// TwinCAT 3 PLC project PLC1
// ProgramVersion: 3.1.4024.12
// libraries:
//   Tc2_EtherCAT, * (Beckhoff Automation GmbH)
//   Tc2_Standard, * (Beckhoff Automation GmbH)
//   Tc2_System, * (Beckhoff Automation GmbH)
//   Tc2_Utilities, * (Beckhoff Automation GmbH)
//   Tc3_Module, * (Beckhoff Automation GmbH)
//   VisuSymbols,3.5.10.0,System
// project tree:
//   / Class Diagram.TcCD (not stored), GlobalTextList.TcGTLO, PlcTask.TcTTO, Visualization Manager.TcVMO (not stored)
//   DUTs/ ST_1In.TcDUT, ST_1In1Out.TcDUT, ST_2In.TcDUT, ST_2Out.TcDUT, ST_EL1004.TcDUT, ST_EL1008.TcDUT, ST_EL2004.TcDUT, ST_EL2008.TcDUT
//   GVLs/ GVL_Constants.TcGVL, GVL_HMI.TcGVL, GVL_IO.TcGVL
//   POUs/FunctionBlocks/ FB_1In.TcPOU, FB_1In_1Out.TcPOU, FB_2In.TcPOU, FB_2Out.TcPOU
//   POUs/FunctionBlocks/Flow FBs/ FB_HandshakeControl.TcPOU
//   POUs/Interfaces/ I_ConveyerSection.TcIO
//   POUs/ MAIN.TcPOU
//   VISUs/ Physical.TcVIS, Configured.TcVIS, RackText.TcTLO
// real-time tasks:
//   TASK PlcTask: cycle T#10ms, priority 20, ADS port 350
//   TASK VISU_TASK: cycle T#200000us, priority 30, ADS port 351
// I/O:
//   DEVICE HotConnect Demo(EtherCAT), AmsNetId 5.29.120.74.5.1
//     2 In_1 [EK1101 EtherCAT Coupler (2A E-Bus, ID switch)]
//       Term 11 (EL1008) [EL1008 8Ch. Dig. Input 24V, 3ms]
//       Term 12 (EL1008) [EL1008 8Ch. Dig. Input 24V, 3ms]
//       Term 1 (EL7031) [EL7031 1Ch. Stepper motor output stage (24V, 1.5A)]
//     2 In_2 [EK1101 EtherCAT Coupler (2A E-Bus, ID switch)]
//       Term 14 (EL1008) [EL1008 8Ch. Dig. Input 24V, 3ms]
//       Term 15 (EL1008) [EL1008 8Ch. Dig. Input 24V, 3ms]
//     1 In 1 out_1 [EK1101 EtherCAT Coupler (2A E-Bus, ID switch)]
//       Term 18 (EL1008) [EL1008 8Ch. Dig. Input 24V, 3ms]
//       Term 19 (EL2008) [EL2008 8Ch. Dig. Output 24V, 0.5A]
//     1 in 1 out_2 [EK1101 EtherCAT Coupler (2A E-Bus, ID switch)]
//       Term 20 (EL1008) [EL1008 8Ch. Dig. Input 24V, 3ms]
//       Term 21 (EL2008) [EL2008 8Ch. Dig. Output 24V, 0.5A]
//     2 Out_1 [EK1101 EtherCAT Coupler (2A E-Bus, ID switch)]
//       Term 24 (EL2008) [EL2008 8Ch. Dig. Output 24V, 0.5A]
//       Term 25 (EL2008) [EL2008 8Ch. Dig. Output 24V, 0.5A]
//     2 Out_2 [EK1101 EtherCAT Coupler (2A E-Bus, ID switch)]
//       Term 26 (EL2008) [EL2008 8Ch. Dig. Output 24V, 0.5A]
//       Term 27 (EL2008) [EL2008 8Ch. Dig. Output 24V, 0.5A]
//     1 In_1 [EK1101 EtherCAT Coupler (2A E-Bus, ID switch)]
//       Term 30 (EL1008) [EL1008 8Ch. Dig. Input 24V, 3ms]
//     1 In_2 [EK1101 EtherCAT Coupler (2A E-Bus, ID switch)]
//       Term 31 (EL1008) [EL1008 8Ch. Dig. Input 24V, 3ms]
// variable links:
//   PLC1/PLC1 Instance <-> HotConnect Demo(EtherCAT)/1 In 1 out_1
//     PlcTask Inputs/GVL_IO.arrIds[2] <-> ID/ID
//     PlcTask Inputs/GVL_IO.arrState[2] <-> InfoData/State
//   PLC1/PLC1 Instance <-> HotConnect Demo(EtherCAT)/1 In 1 out_1/Term 18 (EL1008)
//     PlcTask Inputs/MAIN.arrFb1In1Out[0].stRack.ST_In/Input{1..8} <-> Channel {1..8}/Input  (8 links)
//   PLC1/PLC1 Instance <-> HotConnect Demo(EtherCAT)/1 In 1 out_1/Term 19 (EL2008)
//     PlcTask Outputs/MAIN.arrFb1In1Out[0].stRack.ST_Out/Output{1..8} <-> Channel {1..8}/Output  (8 links)
//   PLC1/PLC1 Instance <-> HotConnect Demo(EtherCAT)/1 In_1
//     PlcTask Inputs/GVL_IO.arrIds[6] <-> ID/ID
//     PlcTask Inputs/GVL_IO.arrState[6] <-> InfoData/State
//   PLC1/PLC1 Instance <-> HotConnect Demo(EtherCAT)/1 In_1/Term 30 (EL1008)
//     PlcTask Inputs/MAIN.arrFb1In[0].stRack.ST_In/Input{1..8} <-> Channel {1..8}/Input  (8 links)
//   PLC1/PLC1 Instance <-> HotConnect Demo(EtherCAT)/1 In_2
//     PlcTask Inputs/GVL_IO.arrIds[7] <-> ID/ID
//     PlcTask Inputs/GVL_IO.arrState[7] <-> InfoData/State
//   PLC1/PLC1 Instance <-> HotConnect Demo(EtherCAT)/1 In_2/Term 31 (EL1008)
//     PlcTask Inputs/MAIN.arrFb1In[1].stRack.ST_In/Input{1..8} <-> Channel {1..8}/Input  (8 links)
//   PLC1/PLC1 Instance <-> HotConnect Demo(EtherCAT)/1 in 1 out_2
//     PlcTask Inputs/GVL_IO.arrIds[3] <-> ID/ID
//     PlcTask Inputs/GVL_IO.arrState[3] <-> InfoData/State
//   PLC1/PLC1 Instance <-> HotConnect Demo(EtherCAT)/1 in 1 out_2/Term 20 (EL1008)
//     PlcTask Inputs/MAIN.arrFb1In1Out[1].stRack.ST_In/Input{1..8} <-> Channel {1..8}/Input  (8 links)
//   PLC1/PLC1 Instance <-> HotConnect Demo(EtherCAT)/1 in 1 out_2/Term 21 (EL2008)
//     PlcTask Outputs/MAIN.arrFb1In1Out[1].stRack.ST_Out/Output{1..8} <-> Channel {1..8}/Output  (8 links)
//   PLC1/PLC1 Instance <-> HotConnect Demo(EtherCAT)/2 In_1
//     PlcTask Inputs/GVL_IO.arrIds[0] <-> ID/ID
//     PlcTask Inputs/GVL_IO.arrState[0] <-> InfoData/State
//   PLC1/PLC1 Instance <-> HotConnect Demo(EtherCAT)/2 In_1/Term 11 (EL1008)
//     PlcTask Inputs/MAIN.arrFb2In[0].stRack.ST_in1/Input{1..8} <-> Channel {1..8}/Input  (8 links)
//   PLC1/PLC1 Instance <-> HotConnect Demo(EtherCAT)/2 In_1/Term 12 (EL1008)
//     PlcTask Inputs/MAIN.arrFb2In[0].stRack.ST_in2/Input{1..8} <-> Channel {1..8}/Input  (8 links)
//   PLC1/PLC1 Instance <-> HotConnect Demo(EtherCAT)/2 In_2
//     PlcTask Inputs/GVL_IO.arrIds[1] <-> ID/ID
//     PlcTask Inputs/GVL_IO.arrState[1] <-> InfoData/State
//   PLC1/PLC1 Instance <-> HotConnect Demo(EtherCAT)/2 In_2/Term 14 (EL1008)
//     PlcTask Inputs/MAIN.arrFb2In[1].stRack.ST_in1/Input{1..8} <-> Channel {1..8}/Input  (8 links)
//   PLC1/PLC1 Instance <-> HotConnect Demo(EtherCAT)/2 In_2/Term 15 (EL1008)
//     PlcTask Inputs/MAIN.arrFb2In[1].stRack.ST_in2/Input{1..8} <-> Channel {1..8}/Input  (8 links)
//   PLC1/PLC1 Instance <-> HotConnect Demo(EtherCAT)/2 Out_1
//     PlcTask Inputs/GVL_IO.arrIds[4] <-> ID/ID
//     PlcTask Inputs/GVL_IO.arrState[4] <-> InfoData/State
//   PLC1/PLC1 Instance <-> HotConnect Demo(EtherCAT)/2 Out_1/Term 24 (EL2008)
//     PlcTask Outputs/MAIN.arrFb2Out[0].stRack.ST_Out1/Output{1..8} <-> Channel {1..8}/Output  (8 links)
//   PLC1/PLC1 Instance <-> HotConnect Demo(EtherCAT)/2 Out_1/Term 25 (EL2008)
//     PlcTask Outputs/MAIN.arrFb2Out[0].stRack.ST_Out2/Output{1..8} <-> Channel {1..8}/Output  (8 links)
//   PLC1/PLC1 Instance <-> HotConnect Demo(EtherCAT)/2 Out_2
//     PlcTask Inputs/GVL_IO.arrIds[5] <-> ID/ID
//     PlcTask Inputs/GVL_IO.arrState[5] <-> InfoData/State
//   PLC1/PLC1 Instance <-> HotConnect Demo(EtherCAT)/2 Out_2/Term 26 (EL2008)
//     PlcTask Outputs/MAIN.arrFb2Out[1].stRack.ST_Out1/Output{1..8} <-> Channel {1..8}/Output  (8 links)
//   PLC1/PLC1 Instance <-> HotConnect Demo(EtherCAT)/2 Out_2/Term 27 (EL2008)
//     PlcTask Outputs/MAIN.arrFb2Out[1].stRack.ST_Out2/Output{1..8} <-> Channel {1..8}/Output  (8 links)

CONFIGURATION PLC1
    RESOURCE PLC ON TwinCAT3
        TASK PlcTask(INTERVAL := T#10ms, PRIORITY := 20);
        PROGRAM MAIN WITH PlcTask : MAIN;
    END_RESOURCE
END_CONFIGURATION

// ---- DUTs/ST_1In.TcDUT
TYPE ST_1In :
STRUCT
	ST_In	AT %I*	: ST_EL1008;
END_STRUCT
END_TYPE

// ---- DUTs/ST_1In1Out.TcDUT
TYPE ST_1In1Out :
STRUCT
	ST_In	AT %I*	: ST_EL1008;
	ST_Out	AT %Q*	: ST_EL2008;
END_STRUCT
END_TYPE

// ---- DUTs/ST_2In.TcDUT
TYPE ST_2In :
STRUCT
	ST_in1	AT %I*: ST_EL1008;
	ST_in2	AT %I*: ST_EL1008;
END_STRUCT
END_TYPE

// ---- DUTs/ST_2Out.TcDUT
TYPE ST_2Out :
STRUCT
	ST_Out1		AT %Q*: ST_EL2008;
	ST_Out2		AT %Q*: ST_EL2008;
END_STRUCT
END_TYPE

// ---- DUTs/ST_EL1004.TcDUT
TYPE ST_EL1004 :
STRUCT
	Inputs	AT %I*	: ARRAY[0..3] OF BOOL;
END_STRUCT
END_TYPE

// ---- DUTs/ST_EL1008.TcDUT
TYPE ST_EL1008 :
STRUCT
	Input1	: BOOL;
	Input2	: BOOL;
	Input3	: BOOL;
	Input4	: BOOL;
	Input5	: BOOL;
	Input6	: BOOL;
	Input7	: BOOL;
	Input8	: BOOL;
END_STRUCT
END_TYPE

// ---- DUTs/ST_EL2004.TcDUT
TYPE ST_EL2004 :
STRUCT
	Outputs	AT %Q*	: ARRAY[0..3] OF BOOL;
END_STRUCT
END_TYPE

// ---- DUTs/ST_EL2008.TcDUT
TYPE ST_EL2008 :
STRUCT
	Output1	: BOOL;
	Output2	: BOOL;
	Output3	: BOOL;
	Output4	: BOOL;
	Output5	: BOOL;
	Output6	: BOOL;
	Output7	: BOOL;
	Output8	: BOOL;
END_STRUCT
END_TYPE

// ---- GVLs/GVL_Constants.TcGVL

VAR_GLOBAL CONSTANT
	nMaxGroups			:	UINT := 8; //The number of HC Groups currently configured in the I/O Tree
	nMax2InGroups		: UINT :=2; //The number of
	nMax1In1OutGroups	: UINT :=2;
	nMax2OutGroups		: UINT :=2;
	nMax1InGroups		: UINT :=2;
	nRange				: UINT := 10;
END_VAR

// ---- GVLs/GVL_HMI.TcGVL
{attribute 'qualified_only'}
VAR_GLOBAL
bType1Present	: BOOL;
bType2Present	: BOOL;
bType3Present	: BOOL;	
bType4Present	: BOOL;

arrPresent			: ARRAY[0..GVL_Constants.nMaxGroups-1] OF BOOL;
arrConnected		: ARRAY[0..GVL_Constants.nMaxGroups-1] OF BOOL;
arrPhysicalIds		: ARRAY[0..nMaxGroups-1] OF UINT;
arrRackNames		: ARRAY[0..nMaxGroups-1] OF INT;
arrTerminalNames	: ARRAY[0..15] OF INT;
arrTerminalData		: ARRAY[0..GVL_Constants.nMaxGroups-1] OF ARRAY[0..15] OF BOOL;
arrPhysicalMissing	: ARRAY[0..GVL_Constants.nMaxGroups-1] OF BOOL;
END_VAR

// ---- GVLs/GVL_IO.TcGVL
{attribute 'qualified_only'}
VAR_GLOBAL
	arrIds	AT %I*: ARRAY[0..GVL_Constants.nMaxgroups-1] OF UINT; //Ids read from I/O->PLC links
	nPresent	: INT; //Number of total Conveyer Groups
	arrState	AT %I*: ARRAY[0..GVL_Constants.nMaxGroups-1] OF UINT; //array of the states of each HC Group
	arrPrevState	: ARRAY[0..GVL_Constants.nMaxGroups-1] OF UINT; //array of previously recorded states for the HC Groups. Updated on Change.
END_VAR

// ---- POUs/Interfaces/I_ConveyerSection.TcIO
INTERFACE I_ConveyerSection EXTENDS __SYSTEM.IQueryInterface

PROPERTY DwnStrmHndShkIn : BOOL
SET
END_SET
END_PROPERTY

PROPERTY DwnStrmHndShkOut : BOOL
GET
END_GET
END_PROPERTY

PROPERTY HMI : ARRAY[0..15] OF BOOL
GET
END_GET
END_PROPERTY

PROPERTY Id : UINT
GET
END_GET
SET
END_SET
END_PROPERTY

PROPERTY Pos : INT
GET
END_GET
SET
END_SET
END_PROPERTY

METHOD  Sequence : BOOL
VAR_INPUT
END_VAR
END_METHOD

METHOD startSequence : BOOL
VAR_INPUT
END_VAR
END_METHOD

METHOD stopSequence : BOOL
VAR_INPUT
END_VAR
END_METHOD

PROPERTY UpStrmHndShkIn : BOOL
SET
END_SET
END_PROPERTY

PROPERTY UpStrmHndShkOut : BOOL
GET
END_GET
END_PROPERTY

END_INTERFACE

// ---- POUs/MAIN.TcPOU
PROGRAM MAIN
VAR
(*
*NOTE: This code is an meant as an example of using Hot Connect to create a project with modular I/O.
*It was written for the purpose of demonstration, and is not meant to be used in a real application.
*)
	//Initialize array of each rack type with a maxium size of configured HC groups that match type
	arrFb2In		: ARRAY[0..GVL_Constants.nMax2InGroups-1] OF FB_2In;
	arrFb1In1Out	: ARRAY[0..GVL_Constants.nMax1In1OutGroups-1] OF FB_1In_1Out;
	arrFb2Out		: ARRAY[0..GVL_Constants.nMax2OutGroups-1] OF FB_2Out;
	arrFb1In		: ARRAY[0..GVL_Constants.nMax1InGroups-1] OF FB_1In;
	//variables representing the current count of each group type found.
	n2InCount		: UINT; //number of connected Type 1 2in groups
	n1In1OutCount	: UINT; //number of connected Type 2 1in 1out groups
	n2OutCount		: UINT;	//number of connected Type 3 2out groups
	n1InCount		: UINT; //number of connected Type 4 1in groups
	//This array will hold each of the function blocks, the Program will execute them in the order they are added to the array,
	// starting with index 1
	iSequences	: ARRAY[0..GVL_Constants.nMaxGroups-1]	OF I_ConveyerSection;
	{attribute 'TcAnalytics'}
	bInit		: BOOL := TRUE;
	{attribute 'TcAnalytics'}
	nCASE		: UINT;
	
	bStop		: BOOL;
	startDelay	: TON;
	bDelay		: BOOL;
	bPulse		: BOOL;
	bReset		: BOOL;
	sequenceDelay	: TP;
	nCount			: INT := 0;
	nScanned		: UINT;
	
	//FBs and Variables for finding the physically found EtherCAT Slaves
	fbGetFound			: FB_EcGetScannedSlaves;
	fbReadCouplerId		: FB_EcPhysicalReadCmd;
	arrEcScannedSlaves	: ARRAY [0..EC_MAX_SLAVES] OF ST_EcSlaveScannedData;
	arrScannedIds		: ARRAY	[0..EC_MAX_SLAVES] OF WORD;
	arrPrevIds			: ARRAY [0..EC_MAX_SLAVES] OF WORD;
	bScanned	: BOOL;
	bFindId		: BOOL;
	bIdBusy		: BOOL;
	bIdError	: BOOL;
	nIdErrId	: UDINT;
	nIdCount	: INT;
	bManRecnct	: BOOL := TRUE;
	FB_HndShk	: FB_HandshakeControl;
	iCompare	: I_ConveyerSection :=0;
END_VAR

CASE nCASE OF
0: //Scan IO for physical slaves.
	//The PLC needs to wait for the I/O to be read by the EtherCAT master before executing code.
	//Otherwise this is a race condition, and the PLC will win, the user will lose.
	startDelay(IN:= TRUE,PT := T#3S,Q=>bDelay);
	IF bDelay THEN
		//Once the PLC has waited long enough, it will get all of the scanned slaves.
		bScanned := getScannedSlaves();	
		bDelay := FALSE;
		bInit := FALSE;
	END_IF
	//IF the PLC get the scanned hardware correctly
	IF bScanned THEN
		//Set our counter and move on to the next case
		nCount := 0;
		nCASE := 1;
	END_IF
1://get the Ids of each scanned coupler to match with linked Ids on the FB level
	// If we have not gone through all of the scanned slaves
	IF nCount < nScanned THEN
		//If the physicalRead has been executed fo the current slave.
		IF getFoundIds(nCount) THEN
			// If the Physical Read is not still busy
			IF NOT bIdBusy THEN
				//Tell the fb to Execute
				bFindId := TRUE; 
			//Otherwise, tell it not to execute
			ELSE
				bFindId := FALSE;
			END_IF
			// If the FB has populated the current array index for Scanned Ids move onto the next Index
			IF arrScannedIds[nIdCount] <> 0 THEN 
				nCount := nCount + 1;
				nIdCount := nIdCount +1;
				IF arrScannedIds[nIdCount] <> arrPrevIds[nIdCount] THEN
					arrPrevIds[nIdCount] := arrScannedIds[nIdCount];
				END_IF
			END_IF
		//If the physical Read FB was not executed for the current slave
		ELSE 
			// move on to the next
			nCount := nCount + 1;
		END_IF
		// IF the scanned slaves have all been read from, or skipped, make sure the most recently read index is not set to 0
	ELSIF arrScannedIds[nIdCount-1] <> 0 THEN 
			nCASE := 2;	
	
	END_IF

2://Initiate the FBs and place them in the iSequences array of interfaces, in order.
	Init_FBs();
	nCount := 0;
	nCASE := 3;
3:
	Start();
	
		nCASE :=4;
	
4://Call the Execution methods of the FBs
//Slow down the execution, so the HMI can keep up
startDelay(IN:= NOT bPulse, PT:= T#500MS, Q=> bPulse);
	IF bPulse THEN
		//Exceute the current FunctionBlock method
		Execution(nCount);
		//mov on to the next function block in the chain
		IF nCount < GVL_IO.nPresent-1 THEN
			nCount := nCount + 1;
		ELSE
			nCount := 0;
		END_IF	
	END_IF;
	IF bStop THEN
		nCASE := 5;
	END_IF
5://Stop all execution
	Stop();
	nCASE := 6;
6:
	IF NOT bStop THEN
		nCASE := 3;
	END_IF
	
END_CASE
IF	bREset THEN 
	nCASE := 0;
	FOR nCount := 0 TO GVL_IO.nPresent-1 DO
		iSequences[nCount] := NULL;
		arrScannedIds[nCount] := 0;
	END_FOR
	GVL_IO.nPresent := 0;
	n1In1OutCount := 0;
	n2InCount	:= 0;
	n1InCount	:= 0;
	n2OutCount	:= 0;
	nIdCount	:= 0;
	nCount		:= 0;
	nScanned	:= 0;
	bReset := FALSE;
	bInit := TRUE;
	bScanned	:= FALSE;
END_IF

IF nCASE >=4 THEN
	checkIoStatus();
	FB_HndShk(arrConveyers := iSequences);
END_IF
updateHMI();

METHOD PRIVATE AddFBtoArray : BOOL
VAR_INPUT
	nextFB	: I_ConveyerSection;
	nIndex	: UINT;
END_VAR
iSequences[GVL_IO.nPresent] := nextFB;
iSequences[GVL_IO.nPresent].Id := GVL_IO.arrIds[nIndex];
iSequences[GVL_IO.nPresent].Pos := GVL_IO.nPresent;
GVL_IO.nPresent := GVL_IO.nPresent +1;
END_METHOD

METHOD checkIoStatus : BOOL
VAR_INPUT
END_VAR

VAR
	nIndex: UINT;
END_VAR
//Since the Id process data of Hotconnect groups do not reset to 0 when disconnected, we need to check the State to see if the HC Group is no longer present.
//If it is no longer present, we need to change the order fo execution for the function blocks
IF NOT bManRecnct THEN
	//For each HC groups state,
	FOR nIndex :=0	TO GVL_Constants.nMaxGroups-1 DO
		//Check if the current State is different from the previous state read.
		IF GVL_IO.arrPrevState[nIndex] <> GVL_IO.arrState[nIndex] THEN
			CASE GVL_IO.arrState[nIndex] OF
			16#101://State: INIT Slave is not present 
			//Report the connect loss, and reset the Function Blocks so the PLC stops executing code for it.			
	
					ADSLOGDINT(msgCtrlMask:= ADSLOG_MSGTYPE_WARN , 
					msgFmtStr:= 'HC Group with Id %d is no longer present. Resetting Function Blocks',
					dintArg:= GVL_IO.arrIds[nIndex]);
					bReset := TRUE;
	
			16#8://State: OP
			//Report the newly connected HC Group, and Reset the Function Blocks so the PLC executes code for it.
	
					ADSLOGDINT(msgCtrlMask:= ADSLOG_MSGTYPE_WARN , 
					msgFmtStr:= 'HC Group with Id %d has been connected mid Process. Resetting Function Blocks',
					dintArg:= GVL_IO.arrIds[nIndex]);
					bReset := TRUE;
	
			END_CASE
			GVL_IO.arrPrevState[nIndex] := GVL_IO.arrState[nIndex];
		END_IF
	END_FOR
END_IF
END_METHOD

METHOD Execution : BOOL
VAR_INPUT
	nCount	: INT;
END_VAR

VAR
	//nCount: INT;
END_VAR
//FOR nCount:= 1 TO GVL_IO.nPresent DO
	iSequences[nCount].Sequence();
//END_FOR
END_METHOD

METHOD getFoundIds : BOOL
VAR_INPUT
	nIndex: INT;
END_VAR

VAR
	
	nEk1101Code	: UDINT := 72166482;
END_VAR
IF arrEcScannedSlaves[nIndex].stSlaveIdentity.productCode = nEK1101Code THEN
	fbReadCouplerId(
		sNetId:= '5.29.120.74.5.1', 
		adp:= arrEcScannedSlaves[nIndex].nAddr, 
		ado:= 16#1000, 
		len:= SIZEOF(arrScannedIds[nIdCount]), 
		eType:= eAdressingType_Fixed, 
		pDstBuf:= ADR(arrScannedIds[nIdCount]), 
		bExecute:= bFindId,
		bBusy => bIdBusy,
		bError => bIdError,
		nErrId => nIdErrId);				
		getFoundIds := TRUE;	
ELSE
	getFoundIds := FALSE;
END_IF
END_METHOD

METHOD getScannedSlaves : BOOL
VAR_INPUT
END_VAR
VAR
	nCounter	: INT;
	
END_VAR
fbGetFound(
	bExecute:= bInit, 
	sNetId:= '5.29.120.74.5.1', 
	pArrEcScannedSlaveInfo:= ADR(arrEcScannedSlaves), 
	cbBufLen:= SIZEOF(arrEcScannedSlaves), 
	tTimeout:= , 
	bBusy=> , 
	bError=> , 
	nErrorId=> , 
	nSlaves=> nScanned);

IF nScanned > 0 THEN
	IF arrEcScannedSlaves[nScanned-1].nAddr > 0 THEN
		getScannedSlaves := TRUE;
		END_IF
END_IF
END_METHOD

METHOD Init_FBs : BOOL
VAR_INPUT
END_VAR
VAR
	nCase		:	UINT;	
	nIdIndex	: 	UINT;
	nIndex		: 	UINT;
	nCopies		:	UINT;
	nModId		: 	UINT;
END_VAR
//For each Id read from the scanned slaves...
FOR nIdIndex := 0 TO nIdCount-1 DO
	//,And For each ID read from the I/O->PLC links...
	FOR nIndex := 0 TO nMaxGroups-1 DO
		//compare the two current Ids and if they match...
		IF arrScannedIds[nIdIndex] = GVL_IO.arrIds[nIndex] THEN
			//The I/O->PLC link Id is used for the switch statement case
			nCase := GVL_IO.arrIds[nIndex];
			//we get the ordered number of the Id, but getting the remainder of it modulo the range for conveyer "types"
			//nRange := 10
			nModId := nCASE MOD nRange;
			//If the remainder is 0, then the Id was the nRange'th of that type
			IF nModId = 0 THEN
				nModId := nRange;			
			END_IF
			//Each case is given a range. Each type of conveyers is given a range, so if the Id is within that range, we will assume it is of that type.
			CASE nCase OF
			1..10: //Range of 2Input type HCGroup
				
				IF GVL_IO.arrState[nIndex] = 8 THEN
					IF n2InCount < nMax2InGroups THEN
						AddFBToArray(arrFb2In[nModId-1],nIndex);
						n2InCount := n2InCount +1;	
					ELSE
						nCase := 1000;
					END_IF
				END_IF
			11..20:// Range of 1 Input 1 Output type HC group
				IF GVL_IO.arrState[nIndex] = 8 THEN
					IF n1In1OutCount < nMax1In1OutGroups THEN
						AddFBToArray(arrFb1In1Out[nModId-1],nIndex);
						n1In1OutCount := n1In1OutCount +1;
					ELSE
						nCase := 1000;
					END_IF
				END_IF
			21..30:// Range of 2 Output type HC group
				IF GVL_IO.arrState[nIndex] = 8 THEN
					IF n2OutCount < nMax2OutGroups THEN
						AddFBToArray(arrFb2Out[nModId-1],nIndex);
						n2OutCount := n2OutCount +1;
					ELSE
						nCase := 1000;
					END_IF
				END_IF
			31..40:// Range of 1 Input type HC Group
				IF GVL_IO.arrState[nIndex] = 8 THEN
					IF n1InCount < nMax1InGroups THEN			
						AddFBToArray(arrFb1In[nModId-1],nIndex);
						n1InCount := n1InCount +1;
					ELSE
						nCase := 1000;
					END_IF
				END_IF
			
			1000://Error
					bReset := TRUE;
			END_CASE
			
		END_IF
		GVL_IO.arrPrevState[nIndex] := GVL_IO.arrState[nIndex];
	END_FOR
END_FOR
END_METHOD

METHOD Start : BOOL
VAR_INPUT
END_VAR
VAR
	nCount	: INT;
END_VAR
//for each function block in the sequence array...
FOR nCount:= 0 TO GVL_IO.nPresent-1 DO
	//call that function block's stopSequence method.
	iSequences[nCount].startSequence();
END_FOR
END_METHOD

METHOD Stop : BOOL
VAR_INPUT
END_VAR

VAR
	nCount: INT;
END_VAR
//for each function block in the sequence array...
FOR nCount:= 0 TO GVL_IO.nPresent-1 DO
	//call that function block's stopSequence method.
	iSequences[nCount].stopSequence();
END_FOR
END_METHOD

METHOD updateHMI : BOOL
VAR_INPUT
END_VAR
VAR
	nCount	: INT;
	nCount2	: INT;
	nPresent : INT := 0;
	nIndex	: INT;
	arrIndexes	: ARRAY[0..nMaxGroups-1] OF INT;
END_VAR
GVL_HMI.bType1Present := FALSE;
GVL_HMI.bType2Present := FALSE;
GVL_HMI.bType3Present := FALSE;
GVL_HMI.bType4Present := FALSE;

//update Configured, and some of Pysical
FOR nCount := 0 TO (GVL_Constants.nMaxGroups - 1)DO	 
		GVL_HMI.arrPresent[nCount] := ((GVL_IO.arrIds[nCount] <> 0) AND (GVL_IO.arrState[nCount] = 16#08));
		IF GVL_HMI.arrPresent[nCount] THEN
			arrIndexes[nPresent] := nCount;
			nPresent := nPresent + 1;
		END_IF
		
		GVL_HMI.arrPhysicalMissing[nCount] := TRUE;
		IF (nCount < GVL_IO.nPresent) AND (__QUERYINTERFACE(iSequences[nCount],iCompare)) THEN
			
			GVL_HMI.arrPhysicalIds[nCount] := iSequences[nCount].Id;
			GVL_HMI.arrTerminalData[nCount]:= iSequences[nCount].HMI;
			GVL_HMI.arrPhysicalMissing[nCount] := FALSE;
		END_IF

	CASE GVL_IO.arrIds[nCount] OF
	
	1..10://Type 1
		IF GVL_HMI.arrPresent[nCount] THEN
			GVL_HMI.bType1Present := TRUE;

		END_IF
	11..20://Type 2
		IF GVL_HMI.arrPresent[nCount] THEN
			GVL_HMI.bType2Present := TRUE;

		END_IF
	21..30://Type 3
		IF GVL_HMI.arrPresent[nCount] THEN
			GVL_HMI.bType3Present := TRUE;
			
		END_IF
	31..40://Type 4	
		IF GVL_HMI.arrPresent[nCount] THEN
			GVL_HMI.bType4Present := TRUE;
			
		END_IF
	END_CASE

END_FOR


//update physical version of HMI
FOR nCount := 0 TO (GVL_IO.nPresent - 1)DO
	GVL_HMI.arrConnected[nCount] := FALSE;
	IF nCount < nPresent THEN
	GVL_HMI.arrConnected[nCount] := ((GVL_HMI.arrPhysicalIds[nCount] <> 0) AND (GVL_HMI.arrPresent[arrIndexes[nCount]]));
	END_IF
	nCount2 := nCount*2;
		CASE GVL_HMI.arrPhysicalIds[nCount] OF
			1..10://Type 1
			GVL_HMI.arrTerminalNames[nCount2] := 6;
			GVL_HMI.arrTerminalNames[nCount2+1] := 6;
			GVL_HMI.arrRackNames[nCount] := 1;
			11..20://Type 2
			GVL_HMI.arrTerminalNames[nCount2] := 6;
			GVL_HMI.arrTerminalNames[nCount2+1] := 5;
			GVL_HMI.arrRackNames[nCount] := 2;
			21..30://Type 3
			GVL_HMI.arrTerminalNames[nCount2] := 5;
			GVL_HMI.arrTerminalNames[nCount2+1] := 5;
			GVL_HMI.arrRackNames[nCount] := 3;
			31..40://Type 4	
			GVL_HMI.arrTerminalNames[nCount2] := 6;
			GVL_HMI.arrTerminalNames[nCount2+1] := 7;
			GVL_HMI.arrRackNames[nCount] := 4;
		END_CASE
		
END_FOR
END_METHOD

END_PROGRAM

// ---- POUs/FunctionBlocks/FB_2In.TcPOU
FUNCTION_BLOCK FB_2In IMPLEMENTS  I_ConveyerSection
VAR_INPUT
END_VAR
VAR_OUTPUT
END_VAR
VAR
	stRack	: ST_2In;
	nStep	: UINT;
	bStart	: BOOL;
	_mDwnStrmHndShkIn	: BOOL;
	_mDwnStrmHndShkOut	: BOOL;
	_mUpStrmHndShkIn	: BOOL;
	_mUpStrmHndShkOut	: BOOL;
	_mId				: UINT;
	_mHMI				: ARRAY[0..15] OF BOOL;
	_mPosition			: INT;
END_VAR

Sequence();


PROPERTY DwnStrmHndShkIn : BOOL
SET
_mDwnStrmHndShkIn := DwnStrmHndShkIn;
END_SET
END_PROPERTY


PROPERTY DwnStrmHndShkOut : BOOL
GET
DwnStrmHndShkOut := _mDwnStrmHndShkOut;
END_GET
END_PROPERTY

{warning 'add property implementation'}
PROPERTY HMI : ARRAY [0..15] OF BOOL
GET
_mHMI[0] := stRack.ST_In1.Input1;
_mHMI[1] := stRack.ST_In1.Input2;
_mHMI[2] := stRack.ST_In1.Input3;
_mHMI[3] := stRack.ST_In1.Input4;
_mHMI[4] := stRack.ST_In1.Input5;
_mHMI[5] := stRack.ST_In1.Input6;
_mHMI[6] := stRack.ST_In1.Input7;
_mHMI[7] := stRack.ST_In1.Input8;
_mHMI[8] := stRack.ST_In2.Input1;
_mHMI[9] := stRack.ST_In2.Input2;
_mHMI[10] := stRack.ST_In2.Input3;
_mHMI[11] := stRack.ST_In2.Input4;
_mHMI[12] := stRack.ST_In2.Input5;
_mHMI[13] := stRack.ST_In2.Input6;
_mHMI[14] := stRack.ST_In2.Input7;
_mHMI[15] := stRack.ST_In2.Input8;
HMI := _mHMI;
END_GET
END_PROPERTY


PROPERTY Id : UINT
GET
Id := _mId;
END_GET
SET
_mId := Id;
END_SET
END_PROPERTY

{warning 'add property implementation'}
PROPERTY Pos : INT
GET
Pos := _mPosition;
END_GET
SET
_mPosition := Pos;
END_SET
END_PROPERTY


METHOD  Sequence : BOOL
IF _mDwnStrmHndShkIn THEN
	stRack.ST_In1.Input1 := TRUE;
	stRack.ST_In1.Input3 := TRUE;
	stRack.ST_In1.Input5 := TRUE;
	stRack.ST_In1.Input7 := TRUE;
END_IF

IF _mUpStrmHndShkIn THEN
	stRack.ST_In1.Input2 := TRUE;
	stRack.ST_In1.Input4 := TRUE;
	stRack.ST_In1.Input6 := TRUE;
	stRack.ST_In1.Input8 := TRUE;
END_IF


THIS^._mDwnStrmHndShkOut := THIS^._mUpStrmHndShkIn;
END_METHOD


METHOD startSequence : BOOL
bStart := TRUE;
END_METHOD


METHOD stopSequence : BOOL
bStart := FALSE;
nStep := 0;
THIS^._mDwnStrmHndShkOut := FALSE;
THIS^._mUpStrmHndShkOut := FALSE;
END_METHOD


PROPERTY UpStrmHndShkIn : BOOL
SET
_mUpStrmHndShkIn := UpStrmHndShkIn;
END_SET
END_PROPERTY


PROPERTY UpStrmHndShkOut : BOOL
GET
END_GET
END_PROPERTY

END_FUNCTION_BLOCK

// ---- POUs/FunctionBlocks/FB_1In_1Out.TcPOU
FUNCTION_BLOCK FB_1In_1Out IMPLEMENTS  I_ConveyerSection
VAR_INPUT
END_VAR
VAR_OUTPUT
END_VAR
VAR
	stRack	: ST_1In1Out;
	nStep	: UINT;
	bStart	: BOOL;
	_mDwnStrmHndShkIn	: BOOL;
	_mDwnStrmHndShkOut	: BOOL;
	_mUpStrmHndShkIn	: BOOL;
	_mUpStrmHndShkOut	: BOOL;
	_mId				: UINT;
	_mHMI				: ARRAY[0..15] OF BOOL;
	_mPosition			: INT;
END_VAR

Sequence();


PROPERTY DwnStrmHndShkIn : BOOL
SET
_mDwnStrmHndShkIn := DwnStrmHndShkIn;
END_SET
END_PROPERTY


PROPERTY DwnStrmHndShkOut : BOOL
GET
DwnStrmHndShkOut := _mDwnStrmHndShkOut;
END_GET
END_PROPERTY

{warning 'add property implementation'}
PROPERTY HMI : ARRAY [0..15] OF BOOL
GET
_mHMI[0] := stRack.ST_In.Input1;
_mHMI[1] := stRack.ST_In.Input2;
_mHMI[2] := stRack.ST_In.Input3;
_mHMI[3] := stRack.ST_In.Input4;
_mHMI[4] := stRack.ST_In.Input5;
_mHMI[5] := stRack.ST_In.Input6;
_mHMI[6] := stRack.ST_In.Input7;
_mHMI[7] := stRack.ST_In.Input8;
_mHMI[8] := stRack.ST_Out.Output1;
_mHMI[9] := stRack.ST_Out.Output2;
_mHMI[10] := stRack.ST_Out.Output3;
_mHMI[11] := stRack.ST_Out.Output4;
_mHMI[12] := stRack.ST_Out.Output5;
_mHMI[13] := stRack.ST_Out.Output6;
_mHMI[14] := stRack.ST_Out.Output7;
_mHMI[15] := stRack.ST_Out.Output8;


HMI := _mHMI;
END_GET
END_PROPERTY


PROPERTY Id : UINT
GET
Id := _mId;
END_GET
SET
_mId := Id;
END_SET
END_PROPERTY

{warning 'add property implementation'}
PROPERTY Pos : INT
GET
Pos := _mPosition;
END_GET
SET
_mPosition := Pos;
END_SET
END_PROPERTY

METHOD Sequence : BOOL
VAR_INPUT
END_VAR
IF bStart THEN
CASE nStep OF
0:
	IF THIS^._mDwnStrmHndShkIn THEN
	stRack.ST_Out.Output1 := NOT stRack.ST_Out.Output1;
	nStep := 1;		
	END_IF
1:
	stRack.ST_Out.Output5 := NOT stRack.ST_Out.Output5;
	THIS^._mUpStrmHndShkOut := TRUE;
	nStep := 2;
2:
	
	stRack.ST_Out.Output4 := NOT stRack.ST_Out.Output4;
	nStep := 3;
3:
	stRack.ST_Out.Output3 := NOT stRack.ST_Out.Output3;
	nStep := 4;
4:	
	stRack.ST_Out.Output5 := NOT stRack.ST_Out.Output5;
	nStep := 5;
5:
	stRack.ST_Out.Output6 := NOT stRack.ST_Out.Output6;
	nStep := 6;
6:
	stRack.ST_Out.Output8 := NOT stRack.ST_Out.Output8;
	nStep := 7;
7:
	stRack.ST_Out.Output7 := NOT stRack.ST_Out.Output7;
	nStep :=0;	
	
END_CASE
END_IF

THIS^._mDwnStrmHndShkOut := THIS^._mUpStrmHndShkIn;
END_METHOD


METHOD startSequence : BOOL
bStart := TRUE;
nStep := 0;
stRack.ST_Out.Output1 := FALSE;
stRack.ST_Out.Output2 := FALSE;
stRack.ST_Out.Output3 := FALSE;
stRack.ST_Out.Output4 := FALSE;
stRack.ST_Out.Output5 := FALSE;
stRack.ST_Out.Output6 := FALSE;
stRack.ST_Out.Output7 := FALSE;
stRack.ST_Out.Output8 := FALSE;
END_METHOD


METHOD stopSequence : BOOL
bStart := FALSE;
nStep := 0;
THIS^._mDwnStrmHndShkOut := FALSE;
THIS^._mUpStrmHndShkOut := FALSE;
END_METHOD


PROPERTY UpStrmHndShkIn : BOOL
SET
_mUpStrmHndShkIn := UpStrmHndShkIn;
END_SET
END_PROPERTY


PROPERTY UpStrmHndShkOut : BOOL
GET
UpStrmHndShkOut	:= _mUpStrmHndShkOut;
END_GET
END_PROPERTY

END_FUNCTION_BLOCK

// ---- POUs/FunctionBlocks/FB_2Out.TcPOU
FUNCTION_BLOCK FB_2Out IMPLEMENTS  I_ConveyerSection
VAR_INPUT
END_VAR
VAR_OUTPUT
END_VAR
VAR
	stRack	: ST_2Out;
	nStep	: UINT;
	bStart	: BOOL;
	_mDwnStrmHndShkIn	: BOOL;
	_mDwnStrmHndShkOut	: BOOL;
	_mUpStrmHndShkIn	: BOOL;
	_mUpStrmHndShkOut	: BOOL;
	_mId				: UINT;
	_mHMI				: ARRAY[0..15] OF BOOL;
	_mPosition			: INT;
END_VAR

Sequence();


PROPERTY DwnStrmHndShkIn : BOOL
SET
_mDwnStrmHndShkIn := DwnStrmHndShkIn;
END_SET
END_PROPERTY


PROPERTY DwnStrmHndShkOut : BOOL
GET
DwnStrmHndShkOut := _mDwnStrmHndShkOut;
END_GET
END_PROPERTY

{warning 'add property implementation'}
PROPERTY HMI : ARRAY [0..15] OF BOOL
GET
_mHMI[0] := stRack.ST_Out1.Output1;
_mHMI[1] := stRack.ST_Out1.Output2;
_mHMI[2] := stRack.ST_Out1.Output3;
_mHMI[3] := stRack.ST_Out1.Output4;
_mHMI[4] := stRack.ST_Out1.Output5;
_mHMI[5] := stRack.ST_Out1.Output6;
_mHMI[6] := stRack.ST_Out1.Output7;
_mHMI[7] := stRack.ST_Out1.Output8;
_mHMI[8] := stRack.ST_Out2.Output1;
_mHMI[9] := stRack.ST_Out2.Output2;
_mHMI[10] := stRack.ST_Out2.Output3;
_mHMI[11] := stRack.ST_Out2.Output4;
_mHMI[12] := stRack.ST_Out2.Output5;
_mHMI[13] := stRack.ST_Out2.Output6;
_mHMI[14] := stRack.ST_Out2.Output7;
_mHMI[15] := stRack.ST_Out2.Output8;

HMI := _mHMI;
END_GET
END_PROPERTY


PROPERTY Id : UINT
GET
Id := _mId;
END_GET
SET
_mId := Id;
END_SET
END_PROPERTY

{warning 'add property implementation'}
PROPERTY Pos : INT
GET
Pos := _mPosition;
END_GET
SET
_mPosition := Pos;
END_SET
END_PROPERTY


METHOD  Sequence : BOOL
IF bStart THEN
CASE nStep OF
0:
	stRack.ST_Out1.Output1 := TRUE;
	stRack.ST_Out2.Output1 := FALSE;
	IF _mDwnStrmHndShkIn THEN
		_mDwnStrmHndShkOut := FALSE;
	END_IF
	IF _mUpStrmHndShkIn THEN
		_mUpStrmHndShkOut := TRUE;
	END_IF
	nStep:=1;
1:
	stRack.ST_Out1.Output3 := TRUE;
	stRack.ST_Out2.Output3 := FALSE;
	IF _mDwnStrmHndShkIn THEN
		_mDwnStrmHndShkOut := TRUE;
	END_IF
		IF _mUpStrmHndShkIn THEN
		_mUpStrmHndShkOut := FALSE;
	END_IF
	nStep := 2;
2:
	stRack.ST_Out1.Output5 := TRUE;
	stRack.ST_Out2.Output5 := FALSE;
	IF _mDwnStrmHndShkIn THEN
		_mDwnStrmHndShkOut := FALSE;
	END_IF
		IF _mUpStrmHndShkIn THEN
		_mUpStrmHndShkOut := TRUE;
	END_IF
	nStep:=3;
3:
	stRack.ST_Out1.Output7 := TRUE;
	stRack.ST_Out2.Output7 := FALSE;
	IF _mDwnStrmHndShkIn THEN
		_mDwnStrmHndShkOut := TRUE;
	END_IF
		IF _mUpStrmHndShkIn THEN
		_mUpStrmHndShkOut := FALSE;
	END_IF
	nStep:=4;
4:
	stRack.ST_Out1.Output2 := TRUE;
	stRack.ST_Out2.Output2 := FALSE;
	IF _mDwnStrmHndShkIn THEN
		_mDwnStrmHndShkOut := FALSE;
	END_IF
		IF _mUpStrmHndShkIn THEN
		_mUpStrmHndShkOut := TRUE;
	END_IF
	nStep:=5;
5:
	stRack.ST_Out1.Output4 := TRUE;
	stRack.ST_Out2.Output4 := FALSE;
	IF _mDwnStrmHndShkIn THEN
		_mDwnStrmHndShkOut := TRUE;
	END_IF
		IF _mUpStrmHndShkIn THEN
		_mUpStrmHndShkOut := FALSE;
	END_IF
	nStep:=6;
6:
	stRack.ST_Out1.Output6 := TRUE;
	stRack.ST_Out2.Output6 := FALSE;
	IF _mDwnStrmHndShkIn THEN
		_mDwnStrmHndShkOut := FALSE;
	END_IF
		IF _mUpStrmHndShkIn THEN
		_mUpStrmHndShkOut := TRUE;
	END_IF
	nStep:=7;
7:
	stRack.ST_Out1.Output8 := TRUE;
	stRack.ST_Out2.Output8 := FALSE;
	IF _mDwnStrmHndShkIn THEN
		_mDwnStrmHndShkOut := TRUE;
	END_IF
		IF _mUpStrmHndShkIn THEN
		_mUpStrmHndShkOut := FALSE;
	END_IF
	nStep:=8;
8:
	stRack.ST_Out1.Output1 := FALSE;
	stRack.ST_Out2.Output1 := TRUE;
	IF _mDwnStrmHndShkIn THEN
		_mDwnStrmHndShkOut := FALSE;
	END_IF
		IF _mUpStrmHndShkIn THEN
		_mUpStrmHndShkOut := TRUE;
	END_IF
	nStep:=9;
9:
	stRack.ST_Out1.Output3 := FALSE;
	stRack.ST_Out2.Output3 := TRUE;
	IF _mDwnStrmHndShkIn THEN
		_mDwnStrmHndShkOut := TRUE;
	END_IF
		IF _mUpStrmHndShkIn THEN
		_mUpStrmHndShkOut := FALSE;
	END_IF
	nStep:=10;
10:
	stRack.ST_Out1.Output5 := FALSE;
	stRack.ST_Out2.Output5 := TRUE;
	IF _mDwnStrmHndShkIn THEN
		_mDwnStrmHndShkOut := FALSE;
	END_IF
		IF _mUpStrmHndShkIn THEN
		_mUpStrmHndShkOut := TRUE;
	END_IF
	nStep:=11;
11:
	stRack.ST_Out1.Output7 := FALSE;
	stRack.ST_Out2.Output7 := TRUE;
	IF _mDwnStrmHndShkIn THEN
		_mDwnStrmHndShkOut := TRUE;
	END_IF
		IF _mUpStrmHndShkIn THEN
		_mUpStrmHndShkOut := FALSE;
	END_IF
	nStep:=12;
12:
	stRack.ST_Out1.Output2 := FALSE;
	stRack.ST_Out2.Output2 := TRUE;
	IF _mDwnStrmHndShkIn THEN
		_mDwnStrmHndShkOut := FALSE;
	END_IF
		IF _mUpStrmHndShkIn THEN
		_mUpStrmHndShkOut := TRUE;
	END_IF
	nStep:=13;
13:
	stRack.ST_Out1.Output4 := FALSE;
	stRack.ST_Out2.Output4 := TRUE;
	IF _mDwnStrmHndShkIn THEN
		_mDwnStrmHndShkOut := TRUE;
	END_IF
	nStep:=14;
14:
	stRack.ST_Out1.Output6 := FALSE;
	stRack.ST_Out2.Output6 := TRUE;
	IF _mDwnStrmHndShkIn THEN
		_mDwnStrmHndShkOut := FALSE;
	END_IF
		IF _mUpStrmHndShkIn THEN
		_mUpStrmHndShkOut := FALSE;
	END_IF
	nStep:=15;
15:
	stRack.ST_Out1.Output8 := FALSE;
	stRack.ST_Out2.Output8 := TRUE;
	IF _mDwnStrmHndShkIn THEN
		_mDwnStrmHndShkOut := TRUE;
	END_IF
		IF _mUpStrmHndShkIn THEN
		_mUpStrmHndShkOut := FALSE;
	END_IF
	nStep:=0;

END_CASE
END_IF

THIS^._mDwnStrmHndShkOut := THIS^._mUpStrmHndShkIn;
END_METHOD


METHOD startSequence : BOOL
bStart := TRUE;
nStep := 0;
stRack.ST_Out1.Output1 := FALSE;
stRack.ST_Out1.Output2 := FALSE;
stRack.ST_Out1.Output3 := FALSE;
stRack.ST_Out1.Output4 := FALSE;
stRack.ST_Out1.Output5 := FALSE;
stRack.ST_Out1.Output6 := FALSE;
stRack.ST_Out1.Output7 := FALSE;
stRack.ST_Out1.Output8 := FALSE;
stRack.ST_Out2.Output1 := FALSE;
stRack.ST_Out2.Output2 := FALSE;
stRack.ST_Out2.Output3 := FALSE;
stRack.ST_Out2.Output4 := FALSE;
stRack.ST_Out2.Output5 := FALSE;
stRack.ST_Out2.Output6 := FALSE;
stRack.ST_Out2.Output7 := FALSE;
stRack.ST_Out2.Output8 := FALSE;
END_METHOD

METHOD stopSequence : BOOL
bStart := FALSE;
nStep :=0;
THIS^._mDwnStrmHndShkOut := FALSE;
THIS^._mUpStrmHndShkOut := FALSE;
END_METHOD


PROPERTY UpStrmHndShkIn : BOOL
SET
_mUpStrmHndShkIn := UpStrmHndShkIn;
END_SET
END_PROPERTY


PROPERTY UpStrmHndShkOut : BOOL
GET
UpStrmHndShkOut	:= _mUpStrmHndShkOut;
END_GET
END_PROPERTY

END_FUNCTION_BLOCK

// ---- POUs/FunctionBlocks/FB_1In.TcPOU
FUNCTION_BLOCK FB_1In IMPLEMENTS  I_ConveyerSection
VAR_INPUT
END_VAR
VAR_OUTPUT
END_VAR
VAR
	stRack	: ST_1In;
	nStep	: UINT;
	bStart	: BOOL;
	_mDwnStrmHndShkIn	: BOOL;
	_mDwnStrmHndShkOut	: BOOL;
	_mUpStrmHndShkIn	: BOOL;
	_mUpStrmHndShkOut	: BOOL;
	_mId				: UINT;
	_mHMI				: ARRAY[0..15] OF BOOL;
	_mPosition			: INT;
END_VAR

Sequence();


PROPERTY DwnStrmHndShkIn : BOOL
SET
_mDwnStrmHndShkIn := DwnStrmHndShkIn;
END_SET
END_PROPERTY


PROPERTY DwnStrmHndShkOut : BOOL
GET
DwnStrmHndShkOut := _mDwnStrmHndShkOut;
END_GET
END_PROPERTY

{warning 'add property implementation'}
PROPERTY HMI : ARRAY [0..15] OF BOOL
GET
_mHMI[0] := stRack.ST_In.Input1;
_mHMI[1] := stRack.ST_In.Input2;
_mHMI[2] := stRack.ST_In.Input3;
_mHMI[3] := stRack.ST_In.Input4;
_mHMI[4] := stRack.ST_In.Input5;
_mHMI[5] := stRack.ST_In.Input6;
_mHMI[6] := stRack.ST_In.Input7;
_mHMI[7] := stRack.ST_In.Input8;

HMI := _mHMI;
END_GET
END_PROPERTY


PROPERTY Id : UINT
GET
Id := _mId;
END_GET
SET
_mId := Id;
END_SET
END_PROPERTY

{warning 'add property implementation'}
PROPERTY Pos : INT
GET
Pos := _mPosition;
END_GET
SET
_mPosition := Pos;
END_SET
END_PROPERTY


METHOD Sequence : BOOL
IF _mDwnStrmHndShkIn THEN
	stRack.ST_In.Input1 := TRUE;
	stRack.ST_In.Input3	:= TRUE;
	stRack.ST_In.Input5	:= TRUE;
	stRack.ST_In.Input7	:= TRUE;
END_IF

IF _mUpStrmHndShkIn THEN
	stRack.ST_In.Input2 := TRUE;
	stRack.ST_In.Input4	:= TRUE;
	stRack.ST_In.Input6	:= TRUE;
	stRack.ST_In.Input8	:= TRUE;
END_IF

THIS^._mDwnStrmHndShkOut := THIS^._mUpStrmHndShkIn;
END_METHOD


METHOD startSequence : BOOL
bStart := TRUE;
END_METHOD


METHOD stopSequence : BOOL
bStart := FALSE;
nStep := 0;
THIS^._mDwnStrmHndShkOut := FALSE;
THIS^._mUpStrmHndShkOut := FALSE;
END_METHOD


PROPERTY UpStrmHndShkIn : BOOL
SET
_mUpStrmHndShkIn := UpStrmHndShkIn;
END_SET
END_PROPERTY


PROPERTY UpStrmHndShkOut : BOOL
GET
UpStrmHndShkOut	:= _mUpStrmHndShkOut;
END_GET
END_PROPERTY

END_FUNCTION_BLOCK

// ---- POUs/FunctionBlocks/Flow FBs/FB_HandshakeControl.TcPOU
FUNCTION_BLOCK FB_HandshakeControl
VAR_INPUT
END_VAR
VAR_OUTPUT
END_VAR
VAR
	nCount: INT;
END_VAR
VAR_IN_OUT
	arrConveyers	: ARRAY[0..nMaxGroups-1] OF I_ConveyerSection;
END_VAR

FOR nCount :=0 TO GVL_IO.nPresent-1 DO
	IF nCount < GVL_IO.nPresent-1 THEN
		arrConveyers[nCount+1].UpStrmHndShkIn  := arrConveyers[nCount].DwnStrmHndShkOut;
	END_IF
	IF nCount > 0 THEN
		arrConveyers[nCount-1].DwnStrmHndShkIn := arrConveyers[nCount].UpStrmHndShkOut;
			
	END_IF
END_FOR

END_FUNCTION_BLOCK

// ---- GlobalTextList.TcGTLO
TEXTLIST GlobalTextList
  341 = '1In1Out_1'
  261 = '1In1Out_2'
  97 = '1In_1'
  200 = '1_In2'
  21 = '2In_1'
  392 = '2In_2'
  775 = '2I_n1'
  510 = '2Out_1'
  403 = '2_In1'
  219 = '2_In2'
  132 = 'Configured Order'
  51 = 'Conveyer Type 1'
  131 = 'Conveyer Type 2'
  374 = 'Conveyer Type 3'
  102 = 'Conveyer Type 4'
  243 = 'Conveyer Type1'
  549 = 'Conveyer Type2'
  797 = 'El1008'
  63 = 'EL1008'
  155 = 'EL2008'
  152 = 'GroupBox'
  910 = 'Id: %d'
  847 = 'MAIN.iSequences[INDEX].Id'
  217 = 'Manual'
  985 = 'Operational Order'
  185 = 'Physical Order'
  682 = 'Pre-Configured Network Pool'
  572 = 'Pre-Configured Networks'
  234 = 'Pre-Configured Pool'
  53 = 'Preconfigured Networks'
  969 = 'Re-Init'
  290 = 'Reinit'
  919 = 'Reset'
  288 = 'Scanned Network'
  339 = 'Stop'
  69 = 'Type 1 No.1: 2 Input'
  223 = 'Type 1 No.2: 2 Input'
  415 = 'Type 1: Long Straight No.1: '
  734 = 'Type 1: Long Straight No.2'
  691 = 'Type 2 No.1: 1  Input, 1 Output'
  622 = 'Type 2 No.2: 1  Input, 1 Output'
  15 = 'Type 2: Curved No.1'
  253 = 'Type 2: Curved No.2'
  446 = 'Type 3 No.1: 2 Output'
  378 = 'Type 3 No.2: 2 Output'
  133 = 'Type 3: Incline No.1'
  920 = 'Type 3: Incline No.2'
  931 = 'Type 3:Incline No.1'
  529 = 'Type 4 No.1: 1 Input'
  512 = 'Type 4 No.2: 1 Input'
  331 = 'Type 4: Decline No.1'
  376 = 'Type 4: Decline No.2'
  235 = 'Type1 No.1: 2 Input'
  110 = 'Type1 No.2: 2 Input'
  938 = 'Type2 No.1: 1  Input, 1 Output'
  838 = 'Type2 No.1: 2 Input1In1Out_1'
  424 = 'Type2 No.2: 1  Input, 1 Output'
  380 = 'Type3 No.1: 2 Output'
  207 = 'Type3 No.2: 2 Output'
END_TEXTLIST

// ---- VISUs/Physical.TcVIS
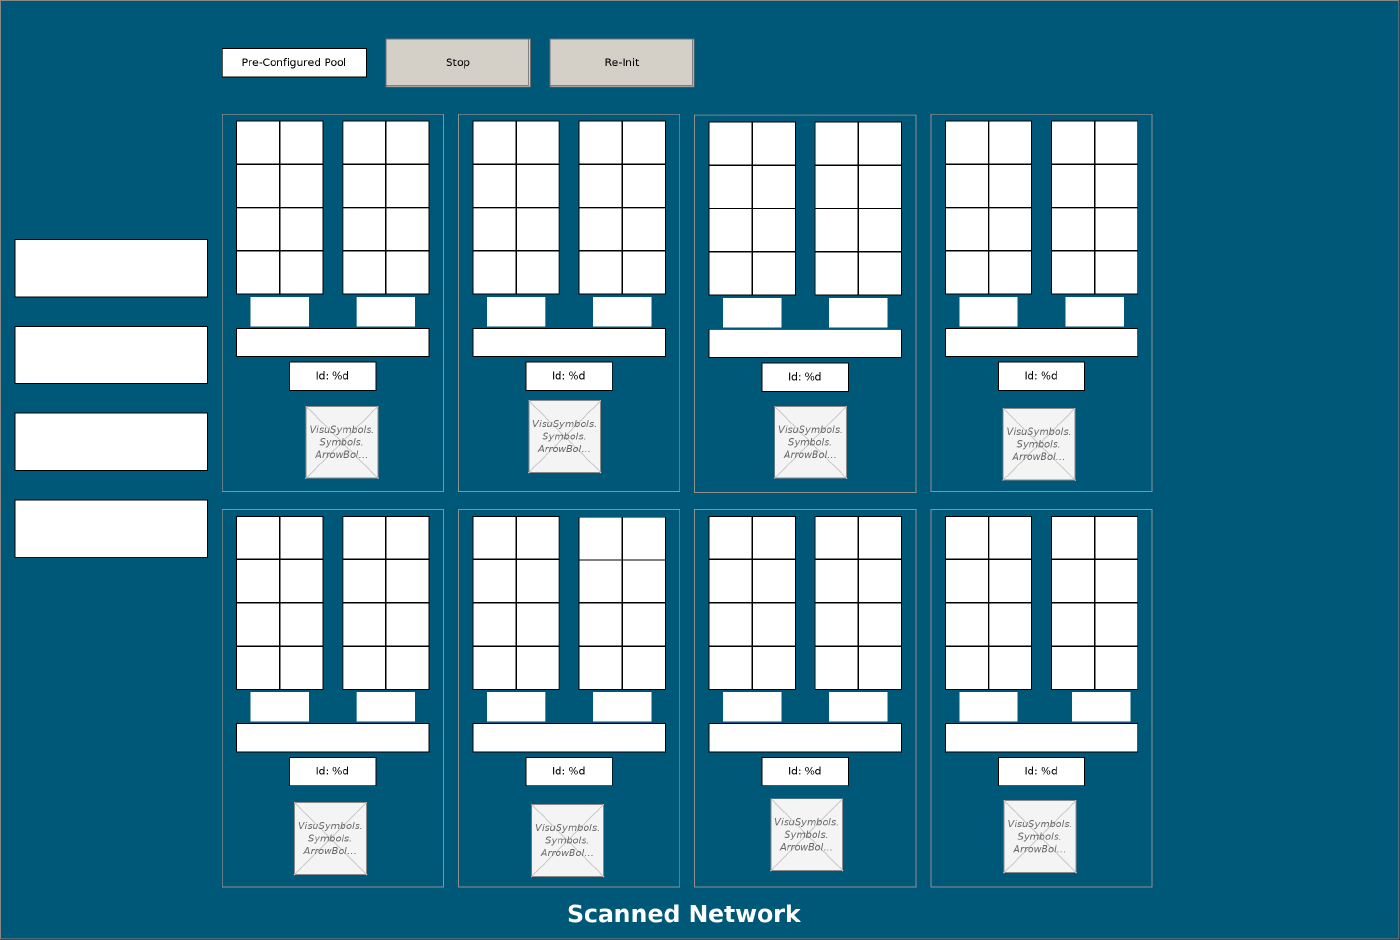
VISUALIZATION Physical  // 1452x975
    RoundedRectangle (0,0 1452x975)
    GroupBox (720,111 230x400), invisible if: GVL_HMI.arrPhysicalMissing[2]
        Rectangle (15,15 45x45), colour toggle: GVL_HMI.arrTerminalData[2][0]
        Rectangle (15,150 45x45), colour toggle: GVL_HMI.arrTerminalData[2][6]
        Rectangle (60,150 45x45), colour toggle: GVL_HMI.arrTerminalData[2][7]
        Rectangle (60,15 45x45), colour toggle: GVL_HMI.arrTerminalData[2][1]
        Rectangle (15,60 45x45), colour toggle: GVL_HMI.arrTerminalData[2][2]
        Rectangle (60,60 45x45), colour toggle: GVL_HMI.arrTerminalData[2][3]
        Rectangle (60,105 45x45), colour toggle: GVL_HMI.arrTerminalData[2][5]
        Rectangle (125,15 45x45), colour toggle: GVL_HMI.arrTerminalData[2][8]
        Rectangle (125,60 45x45), colour toggle: GVL_HMI.arrTerminalData[2][10]
        Rectangle (125,150 45x45), colour toggle: GVL_HMI.arrTerminalData[2][14]
        Rectangle (170,60 45x45), colour toggle: GVL_HMI.arrTerminalData[2][11]
        Rectangle (170,150 45x45), colour toggle: GVL_HMI.arrTerminalData[2][15]
        Rectangle (15,105 45x45), colour toggle: GVL_HMI.arrTerminalData[2][4]
        Rectangle (30,198 60x30), text list: 'RackText', text index: GVL_HMI.arrTerminalNames[4]
        Rectangle (140,198 60x30), text list: 'RackText', text index: GVL_HMI.arrTerminalNames[5]
        Rectangle (170,15 45x45), colour toggle: GVL_HMI.arrTerminalData[2][9]
        Rectangle (125,105 45x45), colour toggle: GVL_HMI.arrTerminalData[2][12]
        Rectangle (170,105 45x45), colour toggle: GVL_HMI.arrTerminalData[2][13]
        Rectangle (70,265 90x30), "Id: %d", text variable: GVL_HMI.arrPhysicalIds[2], colour toggle: GVL_HMI.arrConnected[2]
        Rectangle (15,230 200x30), text list: 'RackText', text index: GVL_HMI.arrRackNames[2]
        Image (83,310 75x75), image: VisuSymbols.Symbols.ArrowBoldRight
    GroupBox (230,520 230x400), invisible if: GVL_HMI.arrPhysicalMissing[4]
        Rectangle (15,15 45x45), colour toggle: GVL_HMI.arrTerminalData[4][0]
        Rectangle (60,15 45x45), colour toggle: GVL_HMI.arrTerminalData[4][1]
        Rectangle (60,105 45x45), colour toggle: GVL_HMI.arrTerminalData[4][5]
        Rectangle (60,150 45x45), colour toggle: GVL_HMI.arrTerminalData[4][7]
        Rectangle (15,60 45x45), colour toggle: GVL_HMI.arrTerminalData[3][2]
        Rectangle (15,105 45x45), colour toggle: GVL_HMI.arrTerminalData[4][4]
        Rectangle (15,150 45x45), colour toggle: GVL_HMI.arrTerminalData[4][6]
        Rectangle (60,60 45x45), colour toggle: GVL_HMI.arrTerminalData[4][3]
        Rectangle (125,15 45x45), colour toggle: GVL_HMI.arrTerminalData[4][8]
        Rectangle (170,15 45x45), colour toggle: GVL_HMI.arrTerminalData[4][9]
        Rectangle (125,60 45x45), colour toggle: GVL_HMI.arrTerminalData[4][10]
        Rectangle (170,60 45x45), colour toggle: GVL_HMI.arrTerminalData[4][11]
        Rectangle (125,105 45x45), colour toggle: GVL_HMI.arrTerminalData[4][12]
        Rectangle (170,105 45x45), colour toggle: GVL_HMI.arrTerminalData[4][13]
        Rectangle (125,150 45x45), colour toggle: GVL_HMI.arrTerminalData[4][14]
        Rectangle (170,150 45x45), colour toggle: GVL_HMI.arrTerminalData[4][15]
        Rectangle (30,198 60x30), text list: 'RackText', text index: GVL_HMI.arrTerminalNames[8]
        Rectangle (140,198 60x30), text list: 'RackText', text index: GVL_HMI.arrTerminalNames[9]
        Rectangle (70,265 90x30), "Id: %d", text variable: GVL_HMI.arrPhysicalIds[4], colour toggle: GVL_HMI.arrConnected[4]
        Rectangle (15,230 200x30), text list: 'RackText', text index: GVL_HMI.arrRackNames[4]
        Image (75,312 75x75), image: VisuSymbols.Symbols.ArrowBoldRight
    GroupBox (475,110 230x400), invisible if: GVL_HMI.arrPhysicalMissing[1]
        Rectangle (15,15 45x45), colour toggle: GVL_HMI.arrTerminalData[1][0]
        Rectangle (60,15 45x45), colour toggle: GVL_HMI.arrTerminalData[1][1]
        Rectangle (60,105 45x45), colour toggle: GVL_HMI.arrTerminalData[1][5]
        Rectangle (60,150 45x45), colour toggle: GVL_HMI.arrTerminalData[1][7]
        Rectangle (15,60 45x45), colour toggle: GVL_HMI.arrTerminalData[1][2]
        Rectangle (15,105 45x45), colour toggle: GVL_HMI.arrTerminalData[1][4]
        Rectangle (15,150 45x45), colour toggle: GVL_HMI.arrTerminalData[1][6]
        Rectangle (60,60 45x45), colour toggle: GVL_HMI.arrTerminalData[1][3]
        Rectangle (125,15 45x45), colour toggle: GVL_HMI.arrTerminalData[1][8]
        Rectangle (170,15 45x45), colour toggle: GVL_HMI.arrTerminalData[1][9]
        Rectangle (125,60 45x45), colour toggle: GVL_HMI.arrTerminalData[1][10]
        Rectangle (170,60 45x45), colour toggle: GVL_HMI.arrTerminalData[1][11]
        Rectangle (125,105 45x45), colour toggle: GVL_HMI.arrTerminalData[1][12]
        Rectangle (170,105 45x45), colour toggle: GVL_HMI.arrTerminalData[1][13]
        Rectangle (125,150 45x45), colour toggle: GVL_HMI.arrTerminalData[1][14]
        Rectangle (170,150 45x45), colour toggle: GVL_HMI.arrTerminalData[1][15]
        Rectangle (30,198 60x30), text list: 'RackText', text index: GVL_HMI.arrTerminalNames[2]
        Rectangle (140,198 60x30), text list: 'RackText', text index: GVL_HMI.arrTerminalNames[3]
        Rectangle (70,265 90x30), "Id: %d", text variable: GVL_HMI.arrPhysicalIds[1], colour toggle: GVL_HMI.arrConnected[1]
        Rectangle (15,230 200x30), text list: 'RackText', text index: GVL_HMI.arrRackNames[1]
        Image (73,305 75x75), image: VisuSymbols.Symbols.ArrowBoldRight
    GroupBox (965,110 230x400), invisible if: GVL_HMI.arrPhysicalMissing[3]
        Rectangle (15,15 45x45), colour toggle: GVL_HMI.arrTerminalData[3][0]
        Rectangle (60,15 45x45), colour toggle: GVL_HMI.arrTerminalData[3][1]
        Rectangle (60,105 45x45), colour toggle: GVL_HMI.arrTerminalData[3][4]
        Rectangle (60,150 45x45), colour toggle: GVL_HMI.arrTerminalData[3][6]
        Rectangle (15,60 45x45), colour toggle: GVL_HMI.arrTerminalData[3][2]
        Rectangle (15,105 45x45), colour toggle: GVL_HMI.arrTerminalData[3][3]
        Rectangle (15,150 45x45), colour toggle: GVL_HMI.arrTerminalData[3][5]
        Rectangle (60,60 45x45), colour toggle: GVL_HMI.arrTerminalData[3][3]
        Rectangle (125,15 45x45), colour toggle: GVL_HMI.arrTerminalData[3][8]
        Rectangle (170,15 45x45), colour toggle: GVL_HMI.arrTerminalData[3][9]
        Rectangle (125,60 45x45), colour toggle: GVL_HMI.arrTerminalData[3][10]
        Rectangle (170,60 45x45), colour toggle: GVL_HMI.arrTerminalData[3][11]
        Rectangle (125,105 45x45), colour toggle: GVL_HMI.arrTerminalData[3][12]
        Rectangle (170,105 45x45), colour toggle: GVL_HMI.arrTerminalData[3][13]
        Rectangle (125,150 45x45), colour toggle: GVL_HMI.arrTerminalData[3][14]
        Rectangle (170,150 45x45), colour toggle: GVL_HMI.arrTerminalData[3][15]
        Rectangle (30,198 60x30), text list: 'RackText', text index: GVL_HMI.arrTerminalNames[6]
        Rectangle (140,198 60x30), text list: 'RackText', text index: GVL_HMI.arrTerminalNames[7]
        Rectangle (70,265 90x30), "Id: %d", text variable: GVL_HMI.arrPhysicalIds[3], colour toggle: GVL_HMI.arrConnected[3]
        Rectangle (15,230 200x30), text list: 'RackText', text index: GVL_HMI.arrRackNames[3]
        Image (75,313 75x75), image: VisuSymbols.Symbols.ArrowBoldRight
    GroupBox (720,520 230x400), invisible if: GVL_HMI.arrPhysicalMissing[6]
        Rectangle (15,15 45x45), colour toggle: MAIN.arrFb1In[0].stRack.ST_In.Input1
        Rectangle (60,15 45x45), colour toggle: MAIN.arrFb1In[0].stRack.ST_In.Input2
        Rectangle (60,105 45x45), colour toggle: MAIN.arrFb1In[0].stRack.ST_In.Input6
        Rectangle (60,150 45x45), colour toggle: MAIN.arrFb1In[0].stRack.ST_In.Input8
        Rectangle (15,60 45x45), colour toggle: MAIN.arrFb1In[0].stRack.ST_In.Input3
        Rectangle (15,105 45x45), colour toggle: MAIN.arrFb1In[0].stRack.ST_In.Input5
        Rectangle (15,150 45x45), colour toggle: MAIN.arrFb1In[0].stRack.ST_In.Input7
        Rectangle (60,60 45x45), colour toggle: MAIN.arrFb1In[0].stRack.ST_In.Input4
        Rectangle (30,198 60x30), text list: 'RackText', text index: GVL_HMI.arrTerminalNames[12]
        Rectangle (70,265 90x30), "Id: %d", text variable: GVL_HMI.arrPhysicalIds[6], colour toggle: GVL_HMI.arrConnected[6]
        Rectangle (125,15 45x45), colour toggle: MAIN.arrFb1In[0].stRack.ST_In.Input1
        Rectangle (140,198 60x30), text list: 'RackText', text index: GVL_HMI.arrTerminalNames[13]
        Rectangle (170,15 45x45), colour toggle: MAIN.arrFb1In[0].stRack.ST_In.Input2
        Rectangle (170,105 45x45), colour toggle: MAIN.arrFb1In[0].stRack.ST_In.Input6
        Rectangle (170,150 45x45), colour toggle: MAIN.arrFb1In[0].stRack.ST_In.Input8
        Rectangle (125,60 45x45), colour toggle: MAIN.arrFb1In[0].stRack.ST_In.Input3
        Rectangle (125,105 45x45), colour toggle: MAIN.arrFb1In[0].stRack.ST_In.Input5
        Rectangle (125,150 45x45), colour toggle: MAIN.arrFb1In[0].stRack.ST_In.Input7
        Rectangle (170,60 45x45), colour toggle: MAIN.arrFb1In[0].stRack.ST_In.Input4
        Rectangle (15,230 200x30), text list: 'RackText', text index: GVL_HMI.arrRackNames[6]
        Image (79,308 75x75), image: VisuSymbols.Symbols.ArrowBoldRight
    GroupBox (230,110 230x400), invisible if: GVL_HMI.arrPhysicalMissing[0]
        Rectangle (15,15 45x45), colour toggle: GVL_HMI.arrTerminalData[0][0]
        Rectangle (60,15 45x45), colour toggle: GVL_HMI.arrTerminalData[0][1]
        Rectangle (60,105 45x45), colour toggle: GVL_HMI.arrTerminalData[0][5]
        Rectangle (60,150 45x45), colour toggle: GVL_HMI.arrTerminalData[0][7]
        Rectangle (15,60 45x45), colour toggle: GVL_HMI.arrTerminalData[0][2]
        Rectangle (15,105 45x45), colour toggle: GVL_HMI.arrTerminalData[0][4]
        Rectangle (15,150 45x45), colour toggle: GVL_HMI.arrTerminalData[0][6]
        Rectangle (60,60 45x45), colour toggle: GVL_HMI.arrTerminalData[0][3]
        Rectangle (125,15 45x45), colour toggle: GVL_HMI.arrTerminalData[0][8]
        Rectangle (125,60 45x45), colour toggle: GVL_HMI.arrTerminalData[0][10]
        Rectangle (170,60 45x45), colour toggle: GVL_HMI.arrTerminalData[0][11]
        Rectangle (125,105 45x45), colour toggle: GVL_HMI.arrTerminalData[0][12]
        Rectangle (170,105 45x45), colour toggle: GVL_HMI.arrTerminalData[0][13]
        Rectangle (125,150 45x45), colour toggle: GVL_HMI.arrTerminalData[0][14]
        Rectangle (170,150 45x45), colour toggle: GVL_HMI.arrTerminalData[0][15]
        Rectangle (30,198 60x30), text list: 'RackText', text index: GVL_HMI.arrTerminalNames[0]
        Rectangle (140,198 60x30), text list: 'RackText', text index: GVL_HMI.arrTerminalNames[1]
        Rectangle (70,265 90x30), "Id: %d", text variable: GVL_HMI.arrPhysicalIds[0], colour toggle: GVL_HMI.arrConnected[0]
        Rectangle (15,230 200x30), text list: 'RackText', text index: GVL_HMI.arrRackNames[0]
        Rectangle (170,15 45x45), colour toggle: GVL_HMI.arrTerminalData[0][9]
        Image (87,311 75x75), image: VisuSymbols.Symbols.ArrowBoldRight
    GroupBox (475,520 230x400), invisible if: GVL_HMI.arrPhysicalMissing[5]
        Rectangle (15,15 45x45), colour toggle: GVL_HMI.arrTerminalData[5][0]
        Rectangle (60,15 45x45), colour toggle: GVL_HMI.arrTerminalData[5][1]
        Rectangle (60,105 45x45), colour toggle: GVL_HMI.arrTerminalData[5][5]
        Rectangle (60,150 45x45), colour toggle: GVL_HMI.arrTerminalData[5][7]
        Rectangle (15,60 45x45), colour toggle: GVL_HMI.arrTerminalData[5][2]
        Rectangle (15,105 45x45), colour toggle: GVL_HMI.arrTerminalData[5][4]
        Rectangle (15,150 45x45), colour toggle: GVL_HMI.arrTerminalData[5][6]
        Rectangle (60,60 45x45), colour toggle: GVL_HMI.arrTerminalData[5][3]
        Rectangle (125,60 45x45), colour toggle: GVL_HMI.arrTerminalData[5][10]
        Rectangle (170,60 45x45), colour toggle: GVL_HMI.arrTerminalData[5][11]
        Rectangle (125,105 45x45), colour toggle: GVL_HMI.arrTerminalData[5][12]
        Rectangle (170,105 45x45), colour toggle: GVL_HMI.arrTerminalData[5][13]
        Rectangle (125,150 45x45), colour toggle: GVL_HMI.arrTerminalData[5][14]
        Rectangle (170,150 45x45), colour toggle: GVL_HMI.arrTerminalData[5][15]
        Rectangle (30,198 60x30), text list: 'RackText', text index: GVL_HMI.arrTerminalNames[10]
        Rectangle (140,198 60x30), text list: 'RackText', text index: GVL_HMI.arrTerminalNames[11]
        Rectangle (170,16 45x45), colour toggle: GVL_HMI.arrTerminalData[5][9]
        Rectangle (125,16 45x45), colour toggle: GVL_HMI.arrTerminalData[5][8]
        Rectangle (70,265 90x30), "Id: %d", text variable: GVL_HMI.arrPhysicalIds[5], colour toggle: GVL_HMI.arrConnected[5]
        Rectangle (15,230 200x30), text list: 'RackText', text index: GVL_HMI.arrRackNames[5]
        Image (76,314 75x75), image: VisuSymbols.Symbols.ArrowBoldRight
    GroupBox (965,520 230x400), invisible if: GVL_HMI.arrPhysicalMissing[7]
        Rectangle (15,15 45x45), colour toggle: MAIN.arrFb1In[1].stRack.ST_In.Input1
        Rectangle (60,15 45x45), colour toggle: MAIN.arrFb1In[1].stRack.ST_In.Input2
        Rectangle (60,105 45x45), colour toggle: MAIN.arrFb1In[1].stRack.ST_In.Input6
        Rectangle (60,150 45x45), colour toggle: MAIN.arrFb1In[1].stRack.ST_In.Input8
        Rectangle (15,60 45x45), colour toggle: MAIN.arrFb1In[1].stRack.ST_In.Input3
        Rectangle (15,105 45x45), colour toggle: MAIN.arrFb1In[1].stRack.ST_In.Input5
        Rectangle (15,150 45x45), colour toggle: MAIN.arrFb1In[1].stRack.ST_In.Input7
        Rectangle (60,60 45x45), colour toggle: MAIN.arrFb1In[1].stRack.ST_In.Input4
        Rectangle (30,198 60x30), text list: 'RackText', text index: GVL_HMI.arrTerminalNames[14]
        Rectangle (70,265 90x30), "Id: %d", text variable: GVL_HMI.arrPhysicalIds[7], colour toggle: GVL_HMI.arrConnected[7]
        Rectangle (125,15 45x45), colour toggle: MAIN.arrFb1In[1].stRack.ST_In.Input1
        Rectangle (147,198 60x30), text list: 'RackText', text index: GVL_HMI.arrTerminalNames[15]
        Rectangle (15,230 200x30), text list: 'RackText', text index: GVL_HMI.arrRackNames[7]
        Rectangle (170,15 45x45), colour toggle: MAIN.arrFb1In[1].stRack.ST_In.Input2
        Rectangle (170,105 45x45), colour toggle: MAIN.arrFb1In[1].stRack.ST_In.Input6
        Rectangle (170,150 45x45), colour toggle: MAIN.arrFb1In[1].stRack.ST_In.Input8
        Rectangle (125,60 45x45), colour toggle: MAIN.arrFb1In[1].stRack.ST_In.Input3
        Rectangle (125,105 45x45), colour toggle: MAIN.arrFb1In[1].stRack.ST_In.Input5
        Rectangle (125,150 45x45), colour toggle: MAIN.arrFb1In[1].stRack.ST_In.Input7
        Rectangle (170,60 45x45), colour toggle: MAIN.arrFb1In[1].stRack.ST_In.Input4
        Image (76,310 75x75), image: VisuSymbols.Symbols.ArrowBoldRight
    Rectangle (230,50 150x30), "Pre-Configured Pool"
        OnMouseDown: change screen: Configured
    Rectangle (15,248 200x60), colour toggle: GVL_HMI.bType1Present, text list: 'RackText', text index: 11
    Rectangle (15,338 200x60), colour toggle: GVL_HMI.bType2Present, text list: 'RackText', text index: 8
    Rectangle (15,428 200x60), colour toggle: GVL_HMI.bType3Present, text list: 'RackText', text index: 9
    Rectangle (15,518 200x60), colour toggle: GVL_HMI.bType4Present, text list: 'RackText', text index: 10
    Button (400,40 150x50), "Stop"
        toggle MAIN.bStop
    Button (570,40 150x50), "Re-Init"
        tap MAIN.bReset
    Label (228,933 963x30), "Scanned Network"
END_VISUALIZATION

// ---- VISUs/Configured.TcVIS
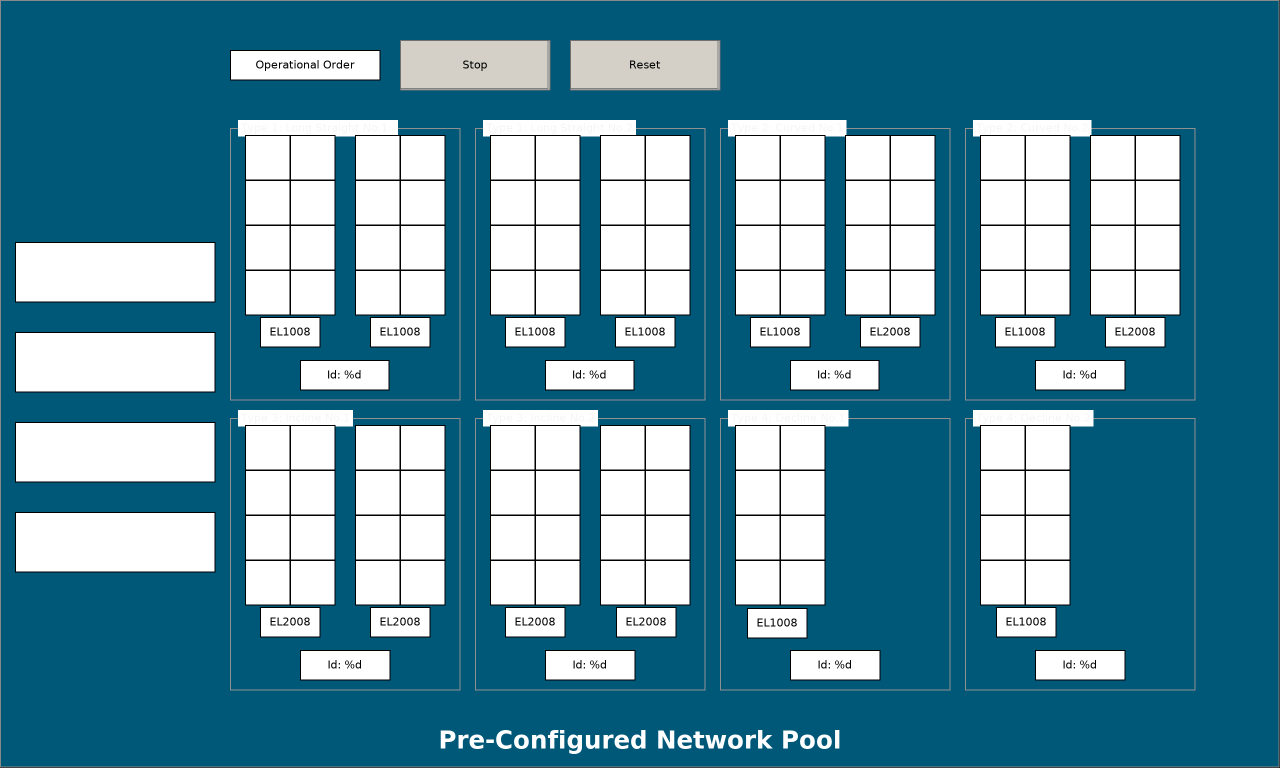
VISUALIZATION Configured  // 1280x768
    RoundedRectangle (0,0 1280x768)
    Rectangle (230,50 150x30), "Operational Order"
        OnMouseDown: change screen: Physical
    Rectangle (15,242 200x60), colour toggle: GVL_HMI.bType1Present, text list: 'RackText', text index: 11
    Rectangle (15,332 200x60), colour toggle: GVL_HMI.bType2Present, text list: 'RackText', text index: 8
    Rectangle (15,422 200x60), colour toggle: GVL_HMI.bType3Present, text list: 'RackText', text index: 9
    Rectangle (15,512 200x60), colour toggle: GVL_HMI.bType4Present, text list: 'RackText', text index: 10
    GroupBox (230,120 230x280), "Type 1: Long Straight No.1:"
        Rectangle (15,15 45x45), colour toggle: MAIN.arrFb2In[0].stRack.ST_in1.Input1
        Rectangle (15,150 45x45), colour toggle: MAIN.arrFb2In[0].stRack.ST_in1.Input7
        Rectangle (60,150 45x45), colour toggle: MAIN.arrFb2In[0].stRack.ST_in1.Input8
        Rectangle (60,15 45x45), colour toggle: MAIN.arrFb2In[0].stRack.ST_in1.Input2
        Rectangle (15,60 45x45), colour toggle: MAIN.arrFb2In[0].stRack.ST_in1.Input3
        Rectangle (60,60 45x45), colour toggle: MAIN.arrFb2In[0].stRack.ST_in1.Input4
        Rectangle (60,105 45x45), colour toggle: MAIN.arrFb2In[0].stRack.ST_in1.Input6
        Rectangle (125,15 45x45), colour toggle: MAIN.arrFb2In[0].stRack.ST_in2.Input1
        Rectangle (125,60 45x45), colour toggle: MAIN.arrFb2In[0].stRack.ST_in2.Input3
        Rectangle (125,150 45x45), colour toggle: MAIN.arrFb2In[0].stRack.ST_in2.Input7
        Rectangle (170,60 45x45), colour toggle: MAIN.arrFb2In[0].stRack.ST_in2.Input4
        Rectangle (170,150 45x45), colour toggle: MAIN.arrFb2In[0].stRack.ST_in2.Input8
        Rectangle (15,105 45x45), colour toggle: MAIN.arrFb2In[0].stRack.ST_in1.Input5
        Rectangle (30,197 60x30), "EL1008"
        Rectangle (140,197 60x30), "EL1008"
        Rectangle (170,15 45x45), colour toggle: MAIN.arrFb2In[0].stRack.ST_in2.Input2
        Rectangle (125,105 45x45), colour toggle: MAIN.arrFb2In[0].stRack.ST_in2.Input5
        Rectangle (170,105 45x45), colour toggle: MAIN.arrFb2In[0].stRack.ST_in2.Input6
        Rectangle (70,240 89x30), "Id: %d", text variable: GVL_IO.arrIds[0], colour toggle: GVL_HMI.arrPresent[0]
    GroupBox (475,120 230x280), "Type 1: Long Straight No.2"
        Rectangle (15,15 45x45), colour toggle: MAIN.arrFb2In[1].stRack.ST_in1.Input1
        Rectangle (60,15 45x45), colour toggle: MAIN.arrFb2In[1].stRack.ST_in1.Input2
        Rectangle (60,105 45x45), colour toggle: MAIN.arrFb2In[1].stRack.ST_in1.Input6
        Rectangle (60,150 45x45), colour toggle: MAIN.arrFb2In[1].stRack.ST_in1.Input8
        Rectangle (15,60 45x45), colour toggle: MAIN.arrFb2In[1].stRack.ST_in1.Input3
        Rectangle (15,105 45x45), colour toggle: MAIN.arrFb2In[1].stRack.ST_in1.Input5
        Rectangle (15,150 45x45), colour toggle: MAIN.arrFb2In[1].stRack.ST_in1.Input7
        Rectangle (60,60 45x45), colour toggle: MAIN.arrFb2In[1].stRack.ST_in1.Input4
        Rectangle (125,15 45x45), colour toggle: MAIN.arrFb2In[1].stRack.ST_in2.Input1
        Rectangle (170,15 45x45), colour toggle: MAIN.arrFb2In[1].stRack.ST_in2.Input2
        Rectangle (125,60 45x45), colour toggle: MAIN.arrFb2In[1].stRack.ST_in2.Input3
        Rectangle (170,60 45x45), colour toggle: MAIN.arrFb2In[1].stRack.ST_in2.Input4
        Rectangle (125,105 45x45), colour toggle: MAIN.arrFb2In[1].stRack.ST_in2.Input5
        Rectangle (170,105 45x45), colour toggle: MAIN.arrFb2In[1].stRack.ST_in2.Input6
        Rectangle (125,150 45x45), colour toggle: MAIN.arrFb2In[1].stRack.ST_in2.Input7
        Rectangle (170,150 45x45), colour toggle: MAIN.arrFb2In[1].stRack.ST_in2.Input8
        Rectangle (30,197 60x30), "EL1008"
        Rectangle (140,197 60x30), "EL1008"
        Rectangle (70,240 89x30), "Id: %d", text variable: GVL_IO.arrIds[1], colour toggle: GVL_HMI.arrPresent[1]
    GroupBox (720,120 230x280), "Type 2: Curved No.1"
        Rectangle (15,15 45x45), colour toggle: MAIN.arrFb1In1Out[0].stRack.ST_In.Input1
        Rectangle (60,15 45x45), colour toggle: MAIN.arrFb1In1Out[0].stRack.ST_In.Input2
        Rectangle (60,105 45x45), colour toggle: MAIN.arrFb1In1Out[0].stRack.ST_In.Input6
        Rectangle (60,150 45x45), colour toggle: MAIN.arrFb1In1Out[0].stRack.ST_In.Input8
        Rectangle (15,60 45x45), colour toggle: MAIN.arrFb1In1Out[0].stRack.ST_In.Input3
        Rectangle (15,105 45x45), colour toggle: MAIN.arrFb1In1Out[0].stRack.ST_In.Input5
        Rectangle (15,150 45x45), colour toggle: MAIN.arrFb1In1Out[0].stRack.ST_In.Input7
        Rectangle (60,60 45x45), colour toggle: MAIN.arrFb1In1Out[0].stRack.ST_In.Input4
        Rectangle (125,15 45x45), colour toggle: MAIN.arrFb1In1Out[0].stRack.ST_Out.Output1
        Rectangle (170,15 45x45), colour toggle: MAIN.arrFb1In1Out[0].stRack.ST_Out.Output2
        Rectangle (125,60 45x45), colour toggle: MAIN.arrFb1In1Out[0].stRack.ST_Out.Output3
        Rectangle (170,60 45x45), colour toggle: MAIN.arrFb1In1Out[0].stRack.ST_Out.Output4
        Rectangle (125,105 45x45), colour toggle: MAIN.arrFb1In1Out[0].stRack.ST_Out.Output5
        Rectangle (170,105 45x45), colour toggle: MAIN.arrFb1In1Out[0].stRack.ST_Out.Output6
        Rectangle (125,150 45x45), colour toggle: MAIN.arrFb1In1Out[0].stRack.ST_Out.Output7
        Rectangle (170,150 45x45), colour toggle: MAIN.arrFb1In1Out[0].stRack.ST_Out.Output8
        Rectangle (30,197 60x30), "EL1008"
        Rectangle (140,197 60x30), "EL2008"
        Rectangle (70,240 89x30), "Id: %d", text variable: GVL_IO.arrIds[2], colour toggle: GVL_HMI.arrPresent[2]
    GroupBox (965,120 230x280), "Type 2: Curved No.2"
        Rectangle (15,15 45x45), colour toggle: MAIN.arrFb1In1Out[1].stRack.ST_In.Input1
        Rectangle (60,15 45x45), colour toggle: MAIN.arrFb1In1Out[1].stRack.ST_In.Input2
        Rectangle (60,105 45x45), colour toggle: MAIN.arrFb1In1Out[1].stRack.ST_In.Input6
        Rectangle (60,150 45x45), colour toggle: MAIN.arrFb1In1Out[1].stRack.ST_In.Input8
        Rectangle (15,60 45x45), colour toggle: MAIN.arrFb1In1Out[1].stRack.ST_In.Input3
        Rectangle (15,105 45x45), colour toggle: MAIN.arrFb1In1Out[1].stRack.ST_In.Input5
        Rectangle (15,150 45x45), colour toggle: MAIN.arrFb1In1Out[1].stRack.ST_In.Input7
        Rectangle (60,60 45x45), colour toggle: MAIN.arrFb1In1Out[1].stRack.ST_In.Input4
        Rectangle (125,15 45x45), colour toggle: MAIN.arrFb1In1Out[1].stRack.ST_Out.Output1
        Rectangle (170,15 45x45), colour toggle: MAIN.arrFb1In1Out[1].stRack.ST_Out.Output2
        Rectangle (125,60 45x45), colour toggle: MAIN.arrFb1In1Out[1].stRack.ST_Out.Output3
        Rectangle (170,60 45x45), colour toggle: MAIN.arrFb1In1Out[1].stRack.ST_Out.Output4
        Rectangle (125,105 45x45), colour toggle: MAIN.arrFb1In1Out[1].stRack.ST_Out.Output5
        Rectangle (170,105 45x45), colour toggle: MAIN.arrFb1In1Out[1].stRack.ST_Out.Output6
        Rectangle (125,150 45x45), colour toggle: MAIN.arrFb1In1Out[1].stRack.ST_Out.Output7
        Rectangle (170,150 45x45), colour toggle: MAIN.arrFb1In1Out[1].stRack.ST_Out.Output8
        Rectangle (30,197 60x30), "EL1008"
        Rectangle (140,197 60x30), "EL2008"
        Rectangle (70,240 90x30), "Id: %d", text variable: GVL_IO.arrIds[3], colour toggle: GVL_HMI.arrPresent[3]
    GroupBox (720,410 230x280), "Type 4: Decline No.1"
        Rectangle (15,15 45x45), colour toggle: MAIN.arrFb1In[0].stRack.ST_In.Input1
        Rectangle (60,15 45x45), colour toggle: MAIN.arrFb1In[0].stRack.ST_In.Input2
        Rectangle (60,105 45x45), colour toggle: MAIN.arrFb1In[0].stRack.ST_In.Input6
        Rectangle (60,150 45x45), colour toggle: MAIN.arrFb1In[0].stRack.ST_In.Input8
        Rectangle (15,60 45x45), colour toggle: MAIN.arrFb1In[0].stRack.ST_In.Input3
        Rectangle (15,105 45x45), colour toggle: MAIN.arrFb1In[0].stRack.ST_In.Input5
        Rectangle (15,150 45x45), colour toggle: MAIN.arrFb1In[0].stRack.ST_In.Input7
        Rectangle (60,60 45x45), colour toggle: MAIN.arrFb1In[0].stRack.ST_In.Input4
        Rectangle (27,198 60x30), "EL1008"
        Rectangle (70,240 90x30), "Id: %d", text variable: GVL_IO.arrIds[6], colour toggle: GVL_HMI.arrPresent[6]
    GroupBox (230,410 230x280), "Type 3: Incline No.1"
        Rectangle (15,15 45x45), colour toggle: MAIN.arrFb2Out[0].stRack.ST_Out1.Output1
        Rectangle (60,15 45x45), colour toggle: MAIN.arrFb2Out[0].stRack.ST_Out1.Output2
        Rectangle (60,105 45x45), colour toggle: MAIN.arrFb2Out[0].stRack.ST_Out1.Output6
        Rectangle (60,150 45x45), colour toggle: MAIN.arrFb2Out[0].stRack.ST_Out1.Output8
        Rectangle (15,60 45x45), colour toggle: MAIN.arrFb2Out[0].stRack.ST_Out1.Output3
        Rectangle (15,105 45x45), colour toggle: MAIN.arrFb2Out[0].stRack.ST_Out1.Output5
        Rectangle (15,150 45x45), colour toggle: MAIN.arrFb2Out[0].stRack.ST_Out1.Output7
        Rectangle (60,60 45x45), colour toggle: MAIN.arrFb2Out[0].stRack.ST_Out1.Output4
        Rectangle (125,15 45x45), colour toggle: MAIN.arrFb2Out[0].stRack.ST_Out2.Output1
        Rectangle (170,15 45x45), colour toggle: MAIN.arrFb2Out[0].stRack.ST_Out2.Output2
        Rectangle (125,60 45x45), colour toggle: MAIN.arrFb2Out[0].stRack.ST_Out2.Output3
        Rectangle (170,60 45x45), colour toggle: MAIN.arrFb2Out[0].stRack.ST_Out2.Output4
        Rectangle (125,105 45x45), colour toggle: MAIN.arrFb2Out[0].stRack.ST_Out2.Output5
        Rectangle (170,105 45x45), colour toggle: MAIN.arrFb2Out[0].stRack.ST_Out2.Output6
        Rectangle (125,150 45x45), colour toggle: MAIN.arrFb2Out[0].stRack.ST_Out2.Output7
        Rectangle (170,150 45x45), colour toggle: MAIN.arrFb2Out[0].stRack.ST_Out2.Output8
        Rectangle (30,197 60x30), "EL2008"
        Rectangle (140,197 60x30), "EL2008"
        Rectangle (70,240 90x30), "Id: %d", text variable: GVL_IO.arrIds[4], colour toggle: GVL_HMI.arrPresent[4]
    GroupBox (475,410 230x280), "Type 3: Incline No.2"
        Rectangle (15,15 45x45), colour toggle: MAIN.arrFb2Out[1].stRack.ST_Out1.Output1
        Rectangle (60,15 45x45), colour toggle: MAIN.arrFb2Out[1].stRack.ST_Out1.Output2
        Rectangle (60,105 45x45), colour toggle: MAIN.arrFb2Out[1].stRack.ST_Out1.Output6
        Rectangle (60,150 45x45), colour toggle: MAIN.arrFb2Out[1].stRack.ST_Out1.Output8
        Rectangle (15,60 45x45), colour toggle: MAIN.arrFb2Out[1].stRack.ST_Out1.Output2
        Rectangle (15,105 45x45), colour toggle: MAIN.arrFb2Out[1].stRack.ST_Out1.Output5
        Rectangle (15,150 45x45), colour toggle: MAIN.arrFb2Out[1].stRack.ST_Out1.Output7
        Rectangle (60,60 45x45), colour toggle: MAIN.arrFb2Out[1].stRack.ST_Out1.Output4
        Rectangle (125,15 45x45), colour toggle: MAIN.arrFb2Out[1].stRack.ST_Out2.Output1
        Rectangle (125,60 45x45), colour toggle: MAIN.arrFb2Out[1].stRack.ST_Out2.Output3
        Rectangle (170,60 45x45), colour toggle: MAIN.arrFb2Out[1].stRack.ST_Out2.Output4
        Rectangle (125,105 45x45), colour toggle: MAIN.arrFb2Out[1].stRack.ST_Out2.Output5
        Rectangle (170,105 45x45), colour toggle: MAIN.arrFb2Out[1].stRack.ST_Out2.Output6
        Rectangle (125,150 45x45), colour toggle: MAIN.arrFb2Out[1].stRack.ST_Out2.Output7
        Rectangle (170,150 45x45), colour toggle: MAIN.arrFb2Out[1].stRack.ST_Out2.Output8
        Rectangle (30,197 60x30), "EL2008"
        Rectangle (141,197 60x30), "EL2008"
        Rectangle (170,15 45x45), colour toggle: MAIN.arrFb2Out[1].stRack.ST_Out2.Output2
        Rectangle (70,240 90x30), "Id: %d", text variable: GVL_IO.arrIds[5], colour toggle: GVL_HMI.arrPresent[5]
    GroupBox (965,410 230x280), "Type 4: Decline No.2"
        Rectangle (15,15 45x45), colour toggle: MAIN.arrFb1In[1].stRack.ST_In.Input1
        Rectangle (60,15 45x45), colour toggle: MAIN.arrFb1In[1].stRack.ST_In.Input2
        Rectangle (60,105 45x45), colour toggle: MAIN.arrFb1In[1].stRack.ST_In.Input6
        Rectangle (60,150 45x45), colour toggle: MAIN.arrFb1In[1].stRack.ST_In.Input8
        Rectangle (15,60 45x45), colour toggle: MAIN.arrFb1In[1].stRack.ST_In.Input3
        Rectangle (15,105 45x45), colour toggle: MAIN.arrFb1In[1].stRack.ST_In.Input5
        Rectangle (15,150 45x45), colour toggle: MAIN.arrFb1In[1].stRack.ST_In.Input7
        Rectangle (60,60 45x45), colour toggle: MAIN.arrFb1In[1].stRack.ST_In.Input4
        Rectangle (31,197 60x30), "EL1008"
        Rectangle (70,240 90x30), "Id: %d", text variable: GVL_IO.arrIds[7], colour toggle: GVL_HMI.arrPresent[7]
    Button (400,40 150x50), "Stop"
        tap MAIN.bStop
    Button (570,40 150x50), "Reset"
        tap MAIN.bReset
    Label (0,725 1280x30), "Pre-Configured Network Pool"
END_VISUALIZATION

// ---- VISUs/RackText.TcTLO
TEXTLIST RackText
  1 = 'Type1: "Long Straight"'
  2 = 'Type2: "Curved"'
  3 = 'Type3:  "Incline"'
  4 = 'Type4: "Decline"'
  5 = 'EL2008'
  6 = 'EL1008'
  7 = 'N/A'
  11 = 'Conveyer Type1: Long Straight: Ids 1-10'
  8 = 'Conveyer Type2: Curved: Ids 11-20'
  9 = 'Conveyer Type3: Incline: Ids 21-30'
  10 = 'Conveyer Type4: Decline: Ids 31-40'
  0 = ''
   = ''
END_TEXTLIST
